            GVL_EVENT.G_Event_Log[GVL_EVENT.G_Event_Head].Event_ID := GVL_EVENT.G_Event_ID_Counter;
GVL_EVENT.G_Event_Log[GVL_EVENT.G_Event_Head].Event_Type := VI_Event_Type;
GVL_EVENT.G_Event_Log[GVL_EVENT.G_Event_Head].Timestamp := VI_Timestamp;
GVL_EVENT.G_Event_Log[GVL_EVENT.G_Event_Head].Param1 := VI_Param1;
GVL_EVENT.G_Event_Log[GVL_EVENT.G_Event_Head].Param2 := VI_Param2;

GVL_EVENT.G_Event_ID_Counter := GVL_EVENT.G_Event_ID_Counter + 1;
GVL_EVENT.G_Event_Head := (GVL_EVENT.G_Event_Head + 1) MOD 64;
          
END_FUNCTION_BLOCK

FUNCTION_BLOCK FB_Fault_Logger
  VAR_INPUT
    VI_Severity : E_System_Severity;
    VI_RootCause : E_System_Root_Cause;
    VI_Time_MS : UDINT;
  END_VAR
  VAR_OUTPUT
    VO_Last_Event_Text : STRING(200);
    VO_Event_Count : UINT;
    VO_Last_Index : UINT;
    VO_Event_Time_MS : ARRAY[1..16] OF UDINT;
    VO_Event_Severity : ARRAY[1..16] OF E_System_Severity;
    VO_Event_RootCause : ARRAY[1..16] OF E_System_Root_Cause;
    VO_Event_Text : ARRAY[1..16] OF STRING(200);
  END_VAR
  VAR
    L_Last_Severity : E_System_Severity;
    L_Last_RootCause : E_System_Root_Cause;
    L_Write_Index : UINT := 0;
    L_Event_Text : STRING(200);
  END_VAR

            L_Event_Text := '';

IF (VI_Severity <> L_Last_Severity) OR (VI_RootCause <> L_Last_RootCause) THEN
    CASE VI_RootCause OF
        E_System_Root_Cause.ROOT_FIRE:
            L_Event_Text := 'EVENT: FIRE DETECTED';
        E_System_Root_Cause.ROOT_GAS_LEAK:
            L_Event_Text := 'EVENT: GAS LEAK';
        E_System_Root_Cause.ROOT_CO_CRITICAL:
            L_Event_Text := 'EVENT: CO CRITICAL';
        E_System_Root_Cause.ROOT_CO_WARNING:
            L_Event_Text := 'EVENT: CO WARNING';
        E_System_Root_Cause.ROOT_WATER_LEAK:
            L_Event_Text := 'EVENT: WATER LEAK';
        E_System_Root_Cause.ROOT_SENSOR_FAULT:
            L_Event_Text := 'EVENT: SENSOR FAULT';
        E_System_Root_Cause.ROOT_IO_OFFLINE:
            L_Event_Text := 'EVENT: IO OFFLINE';
        E_System_Root_Cause.ROOT_COMM_FAULT:
            L_Event_Text := 'EVENT: COMM FAULT';
        E_System_Root_Cause.ROOT_WATCHDOG_FAULT:
            L_Event_Text := 'EVENT: WATCHDOG FAULT';
        E_System_Root_Cause.ROOT_SUBSYSTEM_FAULT:
            L_Event_Text := 'EVENT: SUBSYSTEM FAULT';
        ELSE
            L_Event_Text := 'EVENT: SYSTEM STATE CHANGE';
    END_CASE;

    L_Write_Index := L_Write_Index + 1;
    IF L_Write_Index > 16 THEN
        L_Write_Index := 1;
    END_IF;

    VO_Event_Time_MS[L_Write_Index] := VI_Time_MS;
    VO_Event_Severity[L_Write_Index] := VI_Severity;
    VO_Event_RootCause[L_Write_Index] := VI_RootCause;
    VO_Event_Text[L_Write_Index] := L_Event_Text;

    VO_Last_Index := L_Write_Index;
    VO_Last_Event_Text := L_Event_Text;

    IF VO_Event_Count < 16 THEN
        VO_Event_Count := VO_Event_Count + 1;
    END_IF;
END_IF;

L_Last_Severity := VI_Severity;
L_Last_RootCause := VI_RootCause;
// >>> BULK_SYNC_ANCHOR: FB_Fault_Logger <<<
          
END_FUNCTION_BLOCK

FUNCTION_BLOCK FB_CoreKernel_Live_Observer

            
          
END_FUNCTION_BLOCK

FUNCTION_BLOCK FB_FloorHeating_Overheat_Protection
  VAR_INPUT
    VI_Threshold : REAL := 45.0;
  END_VAR
  VAR_OUTPUT
    VO_Overheat_Detected : BOOL;
    VO_Locked_Circuits : ARRAY[1..GVL_CONSTANTS.C_MAX_HEATING_CIRCUITS] OF BOOL;
  END_VAR
  VAR_IN_OUT
    VI_Temps : ARRAY[1..GVL_CONSTANTS.C_MAX_HEATING_CIRCUITS] OF REAL;
  END_VAR
  VAR
    L_i : INT;
  END_VAR

            VO_Overheat_Detected := FALSE;
FOR L_i := 1 TO GVL_CONSTANTS.C_MAX_HEATING_CIRCUITS DO
    IF VI_Temps[L_i] > VI_Threshold THEN
        VO_Overheat_Detected := TRUE;
        VO_Locked_Circuits[L_i] := TRUE;
    END_IF;
END_FOR;
          
END_FUNCTION_BLOCK

FUNCTION_BLOCK FB_HMI_Interface
  VAR_INPUT
    VI_Severity : E_System_Severity;
    VI_RootCause : E_System_Root_Cause;
    VI_Status_Msg : STRING(200);
  END_VAR
  VAR_OUTPUT
    VO_HMI_Status_Text : STRING(200);
    VO_HMI_State_Code : INT;
  END_VAR

            VO_HMI_Status_Text := VI_Status_Msg;

CASE VI_Severity OF
    E_System_Severity.SEV_NORMAL:
        VO_HMI_State_Code := 0;
    E_System_Severity.SEV_WARNING:
        VO_HMI_State_Code := 1;
    E_System_Severity.SEV_DEGRADED:
        VO_HMI_State_Code := 2;
    E_System_Severity.SEV_CRITICAL:
        VO_HMI_State_Code := 3;
END_CASE;
// >>> BULK_SYNC_ANCHOR: FB_HMI_Interface <<<
          
END_FUNCTION_BLOCK

FUNCTION_BLOCK FB_System_Health
  VAR_INPUT
    VI_Smoke_Detected : BOOL;
    VI_Gas_Detected : BOOL;
    VI_CO_Warning_Level : BOOL;
    VI_CO_Alarm_Level : BOOL;
    VI_Leak_Detected : BOOL;
    VI_Sensor_Fault : BOOL := FALSE;
    VI_IO_Offline : BOOL := FALSE;
    VI_Comm_Fault : BOOL := FALSE;
    VI_Watchdog_Fault : BOOL := FALSE;
    VI_Subsystem_Fault : BOOL := FALSE;
  END_VAR
  VAR_OUTPUT
    VO_System_Severity : E_System_Severity;
    VO_Root_Cause : E_System_Root_Cause;
    VO_Sensor_Fault : BOOL;
    VO_IO_Fault : BOOL;
    VO_Comm_Fault : BOOL;
    VO_Subsystem_Degraded : BOOL;
    VO_First_Fault_Active : BOOL;
    VO_First_Fault_Type : INT;
    VO_First_Fault_Source : INT;
    VO_IO_Fault_Count : UDINT;
    VO_Comm_Fault_Count : UDINT;
    VO_Sensor_Fault_Count : UDINT;
    VO_Subsystem_Fault_Count : UDINT;
    VO_Watchdog_Fault_Count : UDINT;
  END_VAR
  VAR
    L_IO_Fault_Assert_Count : UINT;
    L_IO_Fault_Clear_Count : UINT;
    L_IO_Fault_Stable : BOOL;
    L_Comm_Fault_Assert_Count : UINT;
    L_Comm_Fault_Clear_Count : UINT;
    L_Comm_Fault_Stable : BOOL;
    L_Sensor_Fault_Assert_Count : UINT;
    L_Sensor_Fault_Clear_Count : UINT;
    L_Sensor_Fault_Stable : BOOL;
    L_Subsystem_Assert_Count : UINT;
    L_Subsystem_Clear_Count : UINT;
    L_Subsystem_Fault_Stable : BOOL;
    L_IO_Fault_Prev : BOOL;
    L_Comm_Fault_Prev : BOOL;
    L_Sensor_Fault_Prev : BOOL;
    L_Subsystem_Fault_Prev : BOOL;
    L_Watchdog_Fault_Prev : BOOL;
  END_VAR
  VAR CONSTANT
    C_HEALTH_DEBOUNCE_CYCLES : UINT := 3;
  END_VAR

            // Debounce non-critical diagnostics: require 3 stable cycles to assert/clear
IF VI_IO_Offline THEN
    L_IO_Fault_Clear_Count := 0;
    IF L_IO_Fault_Assert_Count < C_HEALTH_DEBOUNCE_CYCLES THEN
        L_IO_Fault_Assert_Count := L_IO_Fault_Assert_Count + 1;
    END_IF;
    IF L_IO_Fault_Assert_Count >= C_HEALTH_DEBOUNCE_CYCLES THEN
        L_IO_Fault_Stable := TRUE;
    END_IF;
ELSE
    L_IO_Fault_Assert_Count := 0;
    IF L_IO_Fault_Clear_Count < C_HEALTH_DEBOUNCE_CYCLES THEN
        L_IO_Fault_Clear_Count := L_IO_Fault_Clear_Count + 1;
    END_IF;
    IF L_IO_Fault_Clear_Count >= C_HEALTH_DEBOUNCE_CYCLES THEN
        L_IO_Fault_Stable := FALSE;
    END_IF;
END_IF;

IF VI_Comm_Fault THEN
    L_Comm_Fault_Clear_Count := 0;
    IF L_Comm_Fault_Assert_Count < C_HEALTH_DEBOUNCE_CYCLES THEN
        L_Comm_Fault_Assert_Count := L_Comm_Fault_Assert_Count + 1;
    END_IF;
    IF L_Comm_Fault_Assert_Count >= C_HEALTH_DEBOUNCE_CYCLES THEN
        L_Comm_Fault_Stable := TRUE;
    END_IF;
ELSE
    L_Comm_Fault_Assert_Count := 0;
    IF L_Comm_Fault_Clear_Count < C_HEALTH_DEBOUNCE_CYCLES THEN
        L_Comm_Fault_Clear_Count := L_Comm_Fault_Clear_Count + 1;
    END_IF;
    IF L_Comm_Fault_Clear_Count >= C_HEALTH_DEBOUNCE_CYCLES THEN
        L_Comm_Fault_Stable := FALSE;
    END_IF;
END_IF;

IF VI_Sensor_Fault THEN
    L_Sensor_Fault_Clear_Count := 0;
    IF L_Sensor_Fault_Assert_Count < C_HEALTH_DEBOUNCE_CYCLES THEN
        L_Sensor_Fault_Assert_Count := L_Sensor_Fault_Assert_Count + 1;
    END_IF;
    IF L_Sensor_Fault_Assert_Count >= C_HEALTH_DEBOUNCE_CYCLES THEN
        L_Sensor_Fault_Stable := TRUE;
    END_IF;
ELSE
    L_Sensor_Fault_Assert_Count := 0;
    IF L_Sensor_Fault_Clear_Count < C_HEALTH_DEBOUNCE_CYCLES THEN
        L_Sensor_Fault_Clear_Count := L_Sensor_Fault_Clear_Count + 1;
    END_IF;
    IF L_Sensor_Fault_Clear_Count >= C_HEALTH_DEBOUNCE_CYCLES THEN
        L_Sensor_Fault_Stable := FALSE;
    END_IF;
END_IF;

IF VI_Subsystem_Fault THEN
    L_Subsystem_Clear_Count := 0;
    IF L_Subsystem_Assert_Count < C_HEALTH_DEBOUNCE_CYCLES THEN
        L_Subsystem_Assert_Count := L_Subsystem_Assert_Count + 1;
    END_IF;
    IF L_Subsystem_Assert_Count >= C_HEALTH_DEBOUNCE_CYCLES THEN
        L_Subsystem_Fault_Stable := TRUE;
    END_IF;
ELSE
    L_Subsystem_Assert_Count := 0;
    IF L_Subsystem_Clear_Count < C_HEALTH_DEBOUNCE_CYCLES THEN
        L_Subsystem_Clear_Count := L_Subsystem_Clear_Count + 1;
    END_IF;
    IF L_Subsystem_Clear_Count >= C_HEALTH_DEBOUNCE_CYCLES THEN
        L_Subsystem_Fault_Stable := FALSE;
    END_IF;
END_IF;

// Count confirmed fault events on rising edge of stable/critical conditions
IF L_IO_Fault_Stable AND NOT L_IO_Fault_Prev THEN
    VO_IO_Fault_Count := VO_IO_Fault_Count + 1;
END_IF;
L_IO_Fault_Prev := L_IO_Fault_Stable;

IF L_Comm_Fault_Stable AND NOT L_Comm_Fault_Prev THEN
    VO_Comm_Fault_Count := VO_Comm_Fault_Count + 1;
END_IF;
L_Comm_Fault_Prev := L_Comm_Fault_Stable;

IF L_Sensor_Fault_Stable AND NOT L_Sensor_Fault_Prev THEN
    VO_Sensor_Fault_Count := VO_Sensor_Fault_Count + 1;
END_IF;
L_Sensor_Fault_Prev := L_Sensor_Fault_Stable;

IF L_Subsystem_Fault_Stable AND NOT L_Subsystem_Fault_Prev THEN
    VO_Subsystem_Fault_Count := VO_Subsystem_Fault_Count + 1;
END_IF;
L_Subsystem_Fault_Prev := L_Subsystem_Fault_Stable;

IF VI_Watchdog_Fault AND NOT L_Watchdog_Fault_Prev THEN
    VO_Watchdog_Fault_Count := VO_Watchdog_Fault_Count + 1;
END_IF;
L_Watchdog_Fault_Prev := VI_Watchdog_Fault;

VO_Sensor_Fault := L_Sensor_Fault_Stable;
VO_IO_Fault := L_IO_Fault_Stable;
VO_Comm_Fault := L_Comm_Fault_Stable;
VO_Subsystem_Degraded := L_Subsystem_Fault_Stable;

VO_System_Severity := E_System_Severity.SEV_NORMAL;
VO_Root_Cause := E_System_Root_Cause.ROOT_NONE;
VO_First_Fault_Active := FALSE;
VO_First_Fault_Type := 0;
VO_First_Fault_Source := 0;

// Priority: FIRE > GAS > CO > WATER > diagnostics
IF VI_Smoke_Detected THEN
    VO_System_Severity := E_System_Severity.SEV_CRITICAL;
    VO_Root_Cause := E_System_Root_Cause.ROOT_FIRE;
    VO_First_Fault_Active := TRUE;
    VO_First_Fault_Type := 5;

ELSIF VI_Gas_Detected THEN
    VO_System_Severity := E_System_Severity.SEV_CRITICAL;
    VO_Root_Cause := E_System_Root_Cause.ROOT_GAS_LEAK;
    VO_First_Fault_Active := TRUE;
    VO_First_Fault_Type := 6;

ELSIF VI_CO_Alarm_Level THEN
    VO_System_Severity := E_System_Severity.SEV_CRITICAL;
    VO_Root_Cause := E_System_Root_Cause.ROOT_CO_CRITICAL;
    VO_First_Fault_Active := TRUE;
    VO_First_Fault_Type := 7;

ELSIF VI_CO_Warning_Level THEN
    VO_System_Severity := E_System_Severity.SEV_WARNING;
    VO_Root_Cause := E_System_Root_Cause.ROOT_CO_WARNING;
    VO_First_Fault_Active := TRUE;
    VO_First_Fault_Type := 7;

ELSIF VI_Leak_Detected THEN
    VO_System_Severity := E_System_Severity.SEV_WARNING;
    VO_Root_Cause := E_System_Root_Cause.ROOT_WATER_LEAK;
    VO_First_Fault_Active := TRUE;
    VO_First_Fault_Type := 8;

ELSIF VI_Watchdog_Fault THEN
    VO_System_Severity := E_System_Severity.SEV_CRITICAL;
    VO_Root_Cause := E_System_Root_Cause.ROOT_WATCHDOG_FAULT;
    VO_First_Fault_Active := TRUE;
    VO_First_Fault_Type := 9;

ELSIF L_IO_Fault_Stable THEN
    VO_System_Severity := E_System_Severity.SEV_DEGRADED;
    VO_Root_Cause := E_System_Root_Cause.ROOT_IO_OFFLINE;
    VO_First_Fault_Active := TRUE;
    VO_First_Fault_Type := 1;

ELSIF L_Comm_Fault_Stable THEN
    VO_System_Severity := E_System_Severity.SEV_DEGRADED;
    VO_Root_Cause := E_System_Root_Cause.ROOT_COMM_FAULT;
    VO_First_Fault_Active := TRUE;
    VO_First_Fault_Type := 3;

ELSIF L_Sensor_Fault_Stable THEN
    VO_System_Severity := E_System_Severity.SEV_DEGRADED;
    VO_Root_Cause := E_System_Root_Cause.ROOT_SENSOR_FAULT;
    VO_First_Fault_Active := TRUE;
    VO_First_Fault_Type := 2;

ELSIF L_Subsystem_Fault_Stable THEN
    VO_System_Severity := E_System_Severity.SEV_DEGRADED;
    VO_Root_Cause := E_System_Root_Cause.ROOT_SUBSYSTEM_FAULT;
    VO_First_Fault_Active := TRUE;
    VO_First_Fault_Type := 4;
END_IF;
// >>> BULK_SYNC_ANCHOR: FB_System_Health <<<
          
END_FUNCTION_BLOCK

FUNCTION_BLOCK FB_Lifetime_Predictor
  VAR_INPUT
    VI_Runtime_Hours : UDINT;
    VI_Start_Count : UDINT;
    VI_Nominal_Life : UDINT := 10000;
  END_VAR
  VAR_OUTPUT
    VO_Remaining_Percent : BYTE;
    VO_Maintenance_Req : BOOL;
  END_VAR

            // Упрощенная модель износа
IF VI_Nominal_Life > 0 THEN
    VO_Remaining_Percent := TO_BYTE(100 - (VI_Runtime_Hours * 100 / VI_Nominal_Life));
ELSE
    VO_Remaining_Percent := 0;
END_IF;

VO_Maintenance_Req := (VO_Remaining_Percent < 10);
          
END_FUNCTION_BLOCK

FUNCTION_BLOCK FB_Persist_Pipeline
  VAR_INPUT
    VI_PersistStruct : ST_Persist;
    VI_System_Time_MS : UDINT;
    VI_IsActivePLC : BOOL;
  END_VAR
  VAR_OUTPUT
    VO_NVRAM_Cmd : BYTE;
    VO_NVRAM_Offset : UDINT;
    VO_NVRAM_Done : BOOL;
    VO_NVRAM_Err : BOOL;
    VO_NVRAM_ErrID : UDINT;
  END_VAR
  VAR_IN_OUT
    VIO_Apply_Settings : BOOL;
    VIO_Persist_Buffer : ARRAY[0..4] OF BYTE;
    VIO_Last_Written_Persist_Buffer : ARRAY[0..4] OF BYTE;
    VIO_Last_Persist_Write_MS : UDINT;
  END_VAR
  VAR
    fbNVRAMManager : FB_NVRAM_Manager;
    L_Persist_Buffer_Changed : BOOL;
  END_VAR

            // === SERIALIZE PERSIST STRUCT → BUFFER ===

// System Mode
VIO_Persist_Buffer[0] := TO_BYTE(TO_INT(VI_PersistStruct.System_Mode));

// Gas
IF VI_PersistStruct.Safety_Gas_Latched THEN
    VIO_Persist_Buffer[1] := BYTE#1;
ELSE
    VIO_Persist_Buffer[1] := BYTE#0;
END_IF;

// Smoke
IF VI_PersistStruct.Safety_Smoke_Latched THEN
    VIO_Persist_Buffer[2] := BYTE#1;
ELSE
    VIO_Persist_Buffer[2] := BYTE#0;
END_IF;

// Leak
IF VI_PersistStruct.Safety_Leak_Latched THEN
    VIO_Persist_Buffer[3] := BYTE#1;
ELSE
    VIO_Persist_Buffer[3] := BYTE#0;
END_IF;

// DHW Pump
IF VI_PersistStruct.DHW_Heating_Pump THEN
    VIO_Persist_Buffer[4] := BYTE#1;
ELSE
    VIO_Persist_Buffer[4] := BYTE#0;
END_IF;

// === END SERIALIZE ===

L_Persist_Buffer_Changed :=
    (VIO_Persist_Buffer[0] <> VIO_Last_Written_Persist_Buffer[0]) OR
    (VIO_Persist_Buffer[1] <> VIO_Last_Written_Persist_Buffer[1]) OR
    (VIO_Persist_Buffer[2] <> VIO_Last_Written_Persist_Buffer[2]) OR
    (VIO_Persist_Buffer[3] <> VIO_Last_Written_Persist_Buffer[3]) OR
    (VIO_Persist_Buffer[4] <> VIO_Last_Written_Persist_Buffer[4]);

VO_NVRAM_Cmd := 0;
VO_NVRAM_Offset := 0;

IF VIO_Apply_Settings THEN
    // explicit config apply requests a controlled write
    // keep flag set until successful write confirmation
    VO_NVRAM_Cmd := 1;

ELSIF L_Persist_Buffer_Changed THEN
    // controlled write: no more often than once per 60 seconds
    IF (VIO_Last_Persist_Write_MS = 0) OR
       ((VI_System_Time_MS - VIO_Last_Persist_Write_MS) >= 60000) THEN
        VO_NVRAM_Cmd := 1;
    END_IF;
END_IF;

fbNVRAMManager(
    VI_Command := VO_NVRAM_Cmd,
    VI_Offset := VO_NVRAM_Offset,
    VI_DataRef := VIO_Persist_Buffer[0],
    VI_DataSize := 5,
    VI_System_Time_MS := VI_System_Time_MS,
    VI_Operator_ID := 'SYSTEM',
    VI_IsActivePLC := VI_IsActivePLC,
    VI_TwoPersonConfirmation := FALSE,
    VO_Done => VO_NVRAM_Done,
    VO_Error => VO_NVRAM_Err,
    VO_ErrorID => VO_NVRAM_ErrID
);

IF (VO_NVRAM_Cmd = 1) AND VO_NVRAM_Done AND NOT VO_NVRAM_Err THEN
    VIO_Last_Written_Persist_Buffer[0] := VIO_Persist_Buffer[0];
    VIO_Last_Written_Persist_Buffer[1] := VIO_Persist_Buffer[1];
    VIO_Last_Written_Persist_Buffer[2] := VIO_Persist_Buffer[2];
    VIO_Last_Written_Persist_Buffer[3] := VIO_Persist_Buffer[3];
    VIO_Last_Written_Persist_Buffer[4] := VIO_Persist_Buffer[4];
    VIO_Last_Persist_Write_MS := VI_System_Time_MS;
    VIO_Apply_Settings := FALSE;
END_IF;
          
END_FUNCTION_BLOCK

FUNCTION_BLOCK FB_Trend_Adapter
  VAR_INPUT
    VI_Data : ST_Trend_Data;
  END_VAR
  VAR_OUTPUT
    VO_Average : REAL;
    VO_Min : REAL;
    VO_Max : REAL;
    VO_Trend_Up : BOOL;
    VO_Trend_Down : BOOL;
  END_VAR
  VAR
    fbAnalyzer : FB_Trend_Analyzer;
    L_Data_Copy : ARRAY[1..GVL_CONSTANTS.C_MAX_TREND_DATA_POINTS] OF REAL;
    L_Count : INT;
    L_i : INT;
  END_VAR

            // Normalize count to analyzer bounds
L_Count := UDINT_TO_INT(VI_Data.record_count);
IF L_Count < 0 THEN
    L_Count := 0;
END_IF;
IF L_Count > GVL_CONSTANTS.C_MAX_TREND_DATA_POINTS THEN
    L_Count := GVL_CONSTANTS.C_MAX_TREND_DATA_POINTS;
END_IF;

// Copy source values into analyzer-compatible buffer
FOR L_i := 1 TO GVL_CONSTANTS.C_MAX_TREND_DATA_POINTS DO
    L_Data_Copy[L_i] := 0.0;
END_FOR;

IF L_Count > 0 THEN
    FOR L_i := 1 TO L_Count DO
        L_Data_Copy[L_i] := VI_Data.values[L_i];
    END_FOR;
END_IF;

fbAnalyzer(
    VI_Count := L_Count,
    VI_Data := L_Data_Copy,
    VO_Average => VO_Average,
    VO_Max => VO_Max,
    VO_Min => VO_Min,
    VO_Trend_Up => VO_Trend_Up,
    VO_Trend_Down => VO_Trend_Down
);
          
END_FUNCTION_BLOCK

FUNCTION_BLOCK FB_System_Redundancy_Orchestrator
  VAR_IN_OUT
    VIO_Local_State : ST_System_State_Snapshot;
    VIO_Remote_State : ST_System_State_Snapshot;
  END_VAR
  VAR
    fbRedundancy : FB_Redundancy_Manager;
  END_VAR

            // ==============================================================================
// System redundancy orchestrator helper
//
// Internal helper for PRG_System.
// Owns PLC role calculation, heartbeat output projection, and synced-state apply.
// ==============================================================================



// Build local state snapshot for replication.
VIO_Local_State.System_Time_MS := GVL_STATUS.G_System_Time_MS;
VIO_Local_State.Current_Scenario := GVL_STATUS.G_Current_Scenario;
VIO_Local_State.Security_Armed := GVL_ALARM.G_Security_Armed;
VIO_Local_State.Active_Alarms := GVL_ALARM.G_Active_Alarm_Count;
VIO_Local_State.Zone_Valves := GVL_STATE.G_Zone_Valves;
VIO_Local_State.Manifold_Pumps := GVL_STATE.G_Manifold_Pumps;
VIO_Local_State.Lighting_States := GVL_STATE.G_Lighting_Levels;
VIO_Local_State.Blinds_Positions := GVL_STATE.G_Blinds_Positions;
VIO_Local_State.Socket_States := GVL_STATE.G_Socket_States;
VIO_Local_State.Gas_Valve_Closed := GVL_COMMAND.G_Gas_Valve_Close;
VIO_Local_State.Water_Valves_Closed := GVL_COMMAND.G_Close_Valve_36;
VIO_Local_State.Version := VIO_Local_State.Version + 1;

fbRedundancy(
    VI_System_Time_MS := GVL_STATUS.G_System_Time_MS,
    VI_Local_PLC_ID := GVL_STATUS.G_PLC_ID,
    VI_Remote_Pulse := GVL_IO.DI_Partner_Pulse,
    VI_Remote_Is_Active := GVL_IO.DI_Partner_Active,
    VI_Gateway_Ping_OK := GVL_GATEWAY.G_Gateway_Ping_OK,
    VI_Local_State := VIO_Local_State,
    VI_Remote_State := VIO_Remote_State
);

GVL_STATUS.G_Is_Active_PLC := (fbRedundancy.VO_Local_Role = E_PLC_ROLE.ROLE_ACTIVE);
GVL_IO.DO_Heartbeat_Pulse := fbRedundancy.VO_Local_Pulse;
GVL_IO.DO_Active_Status := GVL_STATUS.G_Is_Active_PLC;

IF fbRedundancy.VO_State_Updated THEN
    GVL_STATUS.G_Current_Scenario := fbRedundancy.VO_Synced_State.Current_Scenario;
    GVL_ALARM.G_Security_Armed := fbRedundancy.VO_Synced_State.Security_Armed;
    GVL_STATE.G_Zone_Valves := fbRedundancy.VO_Synced_State.Zone_Valves;
    GVL_STATE.G_Manifold_Pumps := fbRedundancy.VO_Synced_State.Manifold_Pumps;
    GVL_STATE.G_Lighting_Levels := fbRedundancy.VO_Synced_State.Lighting_States;
    GVL_STATE.G_Blinds_Positions := fbRedundancy.VO_Synced_State.Blinds_Positions;
    GVL_STATE.G_Socket_States := fbRedundancy.VO_Synced_State.Socket_States;
    GVL_COMMAND.G_Gas_Valve_Close := fbRedundancy.VO_Synced_State.Gas_Valve_Closed;
    GVL_COMMAND.G_Close_Valve_36 := fbRedundancy.VO_Synced_State.Water_Valves_Closed;
    VIO_Local_State.Version := fbRedundancy.VO_Synced_State.Version;
END_IF;

// >>> BULK_SYNC_ANCHOR: FB_System_Redundancy_Orchestrator <<<
          
END_FUNCTION_BLOCK

FUNCTION_BLOCK FB_Diagnostics_Event_Manager
  VAR_INPUT
    VI_Code : UDINT;
    VI_Severity : INT;
    VI_Active : BOOL;
    VI_Timestamp : UDINT;
    VI_Source : INT;
  END_VAR
  VAR_IN_OUT
    VIO_Events : ARRAY[1..50] OF ST_Diagnostic_Event;
    VIO_Count : INT;
  END_VAR
  VAR
    L_i : INT;
    L_Found_Index : INT;
    L_Was_Active : BOOL;
  END_VAR

            L_Found_Index := 0;
L_Was_Active := FALSE;

FOR L_i := 1 TO VIO_Count DO
    IF (VIO_Events[L_i].Code = VI_Code) AND (VIO_Events[L_i].Source = VI_Source) THEN
        L_Found_Index := L_i;
        L_Was_Active := VIO_Events[L_i].Active;
    END_IF;
END_FOR;

IF VI_Active THEN
    IF L_Found_Index = 0 THEN
        IF VIO_Count < 50 THEN
            VIO_Count := VIO_Count + 1;
            VIO_Events[VIO_Count].Code := VI_Code;
            VIO_Events[VIO_Count].Severity := VI_Severity;
            VIO_Events[VIO_Count].Active := TRUE;
            VIO_Events[VIO_Count].Timestamp := VI_Timestamp;
            VIO_Events[VIO_Count].Source := VI_Source;
        END_IF;
    ELSE
        VIO_Events[L_Found_Index].Severity := VI_Severity;
        IF NOT L_Was_Active THEN
            VIO_Events[L_Found_Index].Timestamp := VI_Timestamp;
        END_IF;
        VIO_Events[L_Found_Index].Active := TRUE;
    END_IF;
ELSE
    IF L_Found_Index > 0 THEN
        VIO_Events[L_Found_Index].Active := FALSE;
    END_IF;
END_IF;
          
END_FUNCTION_BLOCK

FUNCTION_BLOCK FB_Access_Control
  VAR_INPUT
    VI_System_Time_MS : UDINT;
    VI_IsActivePLC : BOOL;
    VI_Armed : BOOL;
    VI_System_Mode : E_System_Operating_Mode;
    VI_Gate_Open_Req : BOOL;
    VI_Wicket_Open_Req : BOOL;
    VI_Lock_1_Open_Req : BOOL;
    VI_Lock_1_Close_Req : BOOL;
    VI_Lock_2_Open_Req : BOOL;
    VI_Lock_2_Close_Req : BOOL;
    VI_PIN_Code : STRING(4);
    VI_RFID_Tag : STRING(20);
    VI_Config : ST_Security_Global_Config;
  END_VAR
  VAR_OUTPUT
    VO_Gate_Open : BOOL;
    VO_Wicket_Open : BOOL;
    VO_Lock_1_Open : BOOL;
    VO_Lock_1_Close : BOOL;
    VO_Lock_2_Open : BOOL;
    VO_Lock_2_Close : BOOL;
  END_VAR
  VAR_IN_OUT
    VI_Access_Codes : ARRAY[1..GVL_CONSTANTS.C_MAX_ACCESS_CODES] OF DWORD;
    VI_RFID_Tags : ARRAY[1..GVL_CONSTANTS.C_MAX_ACCESS_CODES] OF STRING(20);
  END_VAR
  VAR
    L_Gate_Timer : TP;
    L_Wicket_Timer : TP;
    L_Lock_1_Open_T : TP;
    L_Lock_1_Close_T : TP;
    L_Lock_2_Open_T : TP;
    L_Lock_2_Close_T : TP;
    L_Prev_Armed : BOOL;
    L_Auto_Lock_Req : BOOL;
    R_Trig_Gate : R_TRIG;
    R_Trig_Wicket : R_TRIG;
    R_Trig_Lock_1_O : R_TRIG;
    R_Trig_Lock_1_C : R_TRIG;
    R_Trig_Lock_2_O : R_TRIG;
    R_Trig_Lock_2_C : R_TRIG;
    fbAccessCode : FB_AccessCode_Manager;
    L_Valid_PIN : BOOL;
  END_VAR

            // Если ПЛК находится в режиме Standby (резерв), он не должен управлять выходами
IF NOT VI_IsActivePLC THEN
    RETURN;
END_IF;

IF VI_System_Mode = E_System_Operating_Mode.MODE_SAFE_STOP THEN
    VO_Gate_Open := FALSE;
    VO_Wicket_Open := FALSE;
    VO_Lock_1_Open := FALSE;
    VO_Lock_2_Open := FALSE;
    RETURN;
END_IF;

// 1. Логика автоматического закрытия замков при постановке на охрану (ТЗ 3.0)
// При переходе системы в режим "Охрана" принудительно блокируем все замки
IF VI_Armed AND NOT L_Prev_Armed THEN
    L_Auto_Lock_Req := TRUE;
END_IF;
L_Prev_Armed := VI_Armed;

// Детекторы фронта для команд
R_Trig_Gate(CLK := VI_Gate_Open_Req);
R_Trig_Wicket(CLK := VI_Wicket_Open_Req);
R_Trig_Lock_1_O(CLK := VI_Lock_1_Open_Req);
R_Trig_Lock_1_C(CLK := VI_Lock_1_Close_Req OR L_Auto_Lock_Req);
R_Trig_Lock_2_O(CLK := VI_Lock_2_Open_Req);
R_Trig_Lock_2_C(CLK := VI_Lock_2_Close_Req OR L_Auto_Lock_Req);

// Проверка PIN-кода или RFID-метки через менеджер кодов
fbAccessCode(
    VI_System_Time_MS := VI_System_Time_MS,
    VI_IsActivePLC := VI_IsActivePLC,
    VI_Code_To_Check := VI_PIN_Code,
    VI_RFID_To_Check := VI_RFID_Tag,
    VI_Access_Codes := VI_Access_Codes,
    VI_RFID_Tags := VI_RFID_Tags,
    VO_Code_Valid => L_Valid_PIN
);

// 2. Формирование импульсов управления исполнительными механизмами (Pulse Control)
// Открытие ворот и калитки требует валидного ПИН-кода или RFID-метки, если система под охраной
L_Gate_Timer(IN := R_Trig_Gate.Q AND (NOT VI_Armed OR L_Valid_PIN), PT := TO_TIME(VI_Config.gate_open_pulse_ms));
VO_Gate_Open := L_Gate_Timer.Q;

L_Wicket_Timer(IN := R_Trig_Wicket.Q AND (NOT VI_Armed OR L_Valid_PIN), PT := TO_TIME(VI_Config.wicket_open_pulse_ms));
VO_Wicket_Open := L_Wicket_Timer.Q;

L_Lock_1_Open_T(IN := R_Trig_Lock_1_O.Q AND (NOT VI_Armed OR L_Valid_PIN), PT := TO_TIME(VI_Config.lock_open_pulse_ms));
VO_Lock_1_Open := L_Lock_1_Open_T.Q;

L_Lock_1_Close_T(IN := R_Trig_Lock_1_C.Q, PT := TO_TIME(VI_Config.lock_close_pulse_ms));
VO_Lock_1_Close := L_Lock_1_Close_T.Q;

L_Lock_2_Open_T(IN := R_Trig_Lock_2_O.Q AND (NOT VI_Armed OR L_Valid_PIN), PT := TO_TIME(VI_Config.lock_open_pulse_ms));
VO_Lock_2_Open := L_Lock_2_Open_T.Q;

L_Lock_2_Close_T(IN := R_Trig_Lock_2_C.Q, PT := TO_TIME(VI_Config.lock_close_pulse_ms));
VO_Lock_2_Close := L_Lock_2_Close_T.Q;

// Сброс флага автоматического закрытия
IF L_Auto_Lock_Req THEN
    L_Auto_Lock_Req := FALSE;
END_IF;
// >>> BULK_SYNC_ANCHOR: FB_Access_Control <<<
          
END_FUNCTION_BLOCK

FUNCTION_BLOCK FB_Trend_Logger
  VAR_INPUT
    VI_System_Time_MS : UDINT;
    VI_Config : ST_Trend_Config;
    VI_Current_Value : REAL;
  END_VAR
  VAR_OUTPUT
    VO_Data : ST_Trend_Data;
  END_VAR
  VAR
    L_Last_Log_Time : UDINT;
    L_Last_Value : REAL;
    L_Deviation : REAL;
  END_VAR

            IF NOT VI_Config.enabled THEN RETURN; END_IF;

// Логирование по изменению (Deadband) или по времени (раз в час)
L_Deviation := ABS(VI_Current_Value - L_Last_Value);
IF (L_Deviation >= (L_Last_Value * VI_Config.deviation_threshold_percent / 100.0)) OR 
   ((SEL(VI_System_Time_MS >= L_Last_Log_Time, VI_System_Time_MS - L_Last_Log_Time, (4294967295 - L_Last_Log_Time) + VI_System_Time_MS + 1)) >= GVL_CONSTANTS.C_MS_IN_HOUR) THEN
    
    // Запись в массив
    VO_Data.write_index := (VO_Data.record_count MOD 100) + 1;
    VO_Data.values[VO_Data.write_index] := VI_Current_Value;
    VO_Data.timestamps[VO_Data.write_index] := VI_System_Time_MS;

    VO_Data.record_count := VO_Data.record_count + 1;
    VO_Data.sum_values := VO_Data.sum_values + VI_Current_Value;
    
    L_Last_Value := VI_Current_Value;
    L_Last_Log_Time := VI_System_Time_MS;
END_IF;
          
END_FUNCTION_BLOCK

FUNCTION_BLOCK FB_State_Trace_Log
  VAR_INPUT
    VI_System_Time : UDINT;
    VI_Gas_Alarm : BOOL;
    VI_Leak_Alarm : BOOL;
    VI_Pumps : ARRAY[1..4] OF BOOL;
  END_VAR
  VAR_OUTPUT
    VO_Last_Change_Time : UDINT;
  END_VAR
  VAR
    L_Last_Gas : BOOL;
    L_Last_Leak : BOOL;
  END_VAR

            IF (VI_Gas_Alarm <> L_Last_Gas) OR (VI_Leak_Alarm <> L_Last_Leak) THEN
    VO_Last_Change_Time := VI_System_Time;
END_IF;

L_Last_Gas := VI_Gas_Alarm;
L_Last_Leak := VI_Leak_Alarm;
          
END_FUNCTION_BLOCK

FUNCTION_BLOCK FB_System_Timer
  VAR_INPUT
    IN : BOOL;
    PT : TIME;
    VI_System_Time_MS : UDINT;
  END_VAR
  VAR_OUTPUT
    Q : BOOL;
    ET : TIME;
  END_VAR
  VAR
    L_Start_Time : UDINT;
    L_Running : BOOL;
  END_VAR

            // ==============================================================================
// Блок таймера, привязанный к системному времени (System Timer)
// Назначение:
// - Замена стандартного TON для обеспечения точной выдержки времени,
//   независимой от времени цикла ПЛК, с использованием единого системного времени.
// ==============================================================================



IF IN THEN
    IF NOT L_Running THEN
        L_Start_Time := VI_System_Time_MS;
        L_Running := TRUE;
        ET := T#0s;
        Q := FALSE;
    ELSE
        // Обработка переполнения UDINT (примерно 49 дней)
        ET := TO_TIME((SEL(VI_System_Time_MS >= L_Start_Time, VI_System_Time_MS - L_Start_Time, (4294967295 - L_Start_Time) + VI_System_Time_MS + 1)));
        
        IF ET >= PT THEN
            Q := TRUE;
            ET := PT;
        ELSE
            Q := FALSE;
        END_IF;
    END_IF;
ELSE
    L_Running := FALSE;
    ET := T#0s;
    Q := FALSE;
END_IF;
// >>> BULK_SYNC_ANCHOR: FB_System_Timer <<<
          
END_FUNCTION_BLOCK

FUNCTION_BLOCK FB_NVRAM_Manager
  VAR_INPUT
    VI_Command : BYTE;
    VI_Offset : UDINT;
    VI_DataRef : REFERENCE TO BYTE;
    VI_DataSize : UDINT;
    VI_System_Time_MS : UDINT;
    VI_Operator_ID : STRING(10);
    VI_IsActivePLC : BOOL;
    VI_TwoPersonConfirmation : BOOL;
  END_VAR
  VAR_OUTPUT
    VO_Done : BOOL;
    VO_Error : BOOL;
    VO_ErrorID : UDINT;
    VO_HMI_Status_Message : STRING(200);
  END_VAR
  VAR
    L_prev_Command : BYTE;
    L_cmd_rising : BOOL;
    L_i : UDINT;
    L_Data_Changed : BOOL;
    L_pData : POINTER TO BYTE;
  END_VAR
  VAR CONSTANT
    C_MAX_NVRAM_SIZE : UDINT := 12800;
  END_VAR

            // Детекция фронта команды
L_cmd_rising := (VI_Command <> 0) AND (L_prev_Command = 0);
L_prev_Command := VI_Command;

IF L_cmd_rising THEN
    VO_Done := FALSE;
    VO_Error := FALSE;
    VO_ErrorID := 0;
    VO_HMI_Status_Message := '';
    
    // Валидация смещения
    IF VI_Offset >= C_MAX_NVRAM_SIZE THEN
        VO_Error := TRUE;
        VO_ErrorID := 16#1501;
        VO_HMI_Status_Message := 'NVRAM: Неверное смещение';
        VO_Done := TRUE;
        RETURN;
    END_IF;

    // Валидация указателя
    IF NOT __ISVALIDREF(VI_DataRef) THEN
        VO_Error := TRUE;
        VO_ErrorID := 16#150A;
        VO_HMI_Status_Message := 'NVRAM: Недействительная ссылка на данные';
        VO_Done := TRUE;
        RETURN;
    END_IF;

    L_pData := ADR(VI_DataRef);

    IF (VI_Offset + VI_DataSize) > C_MAX_NVRAM_SIZE THEN
        VO_Error := TRUE;
        VO_ErrorID := 16#150B;
        VO_HMI_Status_Message := 'NVRAM: Размер данных превышает доступный объем';
        VO_Done := TRUE;
        RETURN;
    END_IF;

    IF VI_Command = 2 THEN
    VO_Error := TRUE;
    VO_ErrorID := 16#150D;
    VO_HMI_Status_Message := 'NVRAM: READ not implemented';
    VO_Done := TRUE;
    RETURN;
END_IF;

IF VI_Command = 1 THEN // ЗАПИСЬ (WRITE)
        IF NOT VI_IsActivePLC THEN
            VO_Error := TRUE;
            VO_ErrorID := 16#1509;
            VO_HMI_Status_Message := 'NVRAM: Запись запрещена (STANDBY)';
        ELSE
            // Проверка на изменение данных перед записью
            L_Data_Changed := FALSE;
            FOR L_i := 0 TO VI_DataSize - 1 DO
                IF GVL_Retain.G_NVRAM_Data[VI_Offset + L_i] <> L_pData[L_i] THEN
                    L_Data_Changed := TRUE;
                    EXIT;
                END_IF;
            END_FOR;
            
            IF L_Data_Changed THEN
                // Безопасное копирование (WRITE)
                FOR L_i := 0 TO VI_DataSize - 1 DO
                    GVL_Retain.G_NVRAM_Data[VI_Offset + L_i] := L_pData[L_i];
                END_FOR;
                VO_HMI_Status_Message := 'NVRAM: Данные успешно сохранены в RETAIN';
            ELSE
                VO_HMI_Status_Message := 'NVRAM: Данные не изменились, запись пропущена';
            END_IF;
        END_IF;
        VO_Done := TRUE;
    END_IF;
END_IF;

IF VI_Command = 0 THEN
    VO_Done := FALSE;
END_IF;
// >>> BULK_SYNC_ANCHOR: FB_NVRAM_Manager <<<
          
END_FUNCTION_BLOCK

FUNCTION_BLOCK FB_History_Manager
  VAR_INPUT
    VI_System_Time_MS : UDINT;
    VI_Write_Event : BOOL;
    VI_Event : ST_History_Record;
  END_VAR
  VAR_OUTPUT
    VO_Total_Events : UDINT;
  END_VAR
  VAR
    L_Prev_Write_Event : BOOL;
  END_VAR

            IF VI_Write_Event AND NOT L_Prev_Write_Event THEN
    GVL_Retain.G_History_Buffer[GVL_Retain.G_History_Write_Idx] := VI_Event;
    GVL_Retain.G_History_Buffer[GVL_Retain.G_History_Write_Idx].timestamp_ms := VI_System_Time_MS;
    
    GVL_Retain.G_History_Write_Idx := (GVL_Retain.G_History_Write_Idx MOD GVL_CONSTANTS.C_MAX_HISTORY_RECORDS) + 1;
    GVL_Retain.G_History_Total_Events := GVL_Retain.G_History_Total_Events + 1;
END_IF;
L_Prev_Write_Event := VI_Write_Event;

VO_Total_Events := GVL_Retain.G_History_Total_Events;
// >>> BULK_SYNC_ANCHOR: FB_History_Manager <<<
          
END_FUNCTION_BLOCK

FUNCTION_BLOCK FB_Heating_Manifold_Control
  VAR_INPUT
    VI_System_Time_MS : UDINT;
    VI_IsActivePLC : BOOL;
    VI_DHW_Heating_Demand : BOOL;
    VI_Freeze_Mode_Active : BOOL;
    VI_Target_Supply_Temp : REAL;
    VI_Any_Zone_Active : ARRAY[1..GVL_CONSTANTS.C_MAX_MANIFOLDS] OF BOOL;
  END_VAR
  VAR_OUTPUT
    VO_Manifold_Pumps : ARRAY[1..GVL_CONSTANTS.C_MAX_MANIFOLDS] OF BOOL;
    VO_Manifold_Valves : ARRAY[1..GVL_CONSTANTS.C_MAX_MANIFOLDS] OF REAL;
    VO_Status : ARRAY[1..GVL_CONSTANTS.C_MAX_MANIFOLDS] OF ST_Manifold_Status;
  END_VAR
  VAR_IN_OUT
    VI_Manifold_Pressures : ARRAY[1..GVL_CONSTANTS.C_MAX_MANIFOLDS] OF REAL;
    VI_Manifold_Currents : ARRAY[1..GVL_CONSTANTS.C_MAX_MANIFOLDS] OF REAL;
    VI_Manifold_Temps_Supply : ARRAY[1..GVL_CONSTANTS.C_MAX_MANIFOLDS] OF REAL;
    VI_Manifold_Temps_Return : ARRAY[1..GVL_CONSTANTS.C_MAX_MANIFOLDS] OF REAL;
  END_VAR
  VAR
    L_i : INT;
    L_Delta_T : REAL;
    L_PID_Valves : ARRAY[1..GVL_CONSTANTS.C_MAX_MANIFOLDS] OF FB_PID_Controller;
    L_PID_Timer : ARRAY[1..GVL_CONSTANTS.C_MAX_MANIFOLDS] OF FB_System_Timer;
    L_Pump_Run_Timer : ARRAY[1..GVL_CONSTANTS.C_MAX_MANIFOLDS] OF FB_System_Timer;
    L_Pump_Pause_Timer : ARRAY[1..GVL_CONSTANTS.C_MAX_MANIFOLDS] OF FB_System_Timer;
    L_Pump_In_Pause : ARRAY[1..GVL_CONSTANTS.C_MAX_MANIFOLDS] OF BOOL;
    L_Pump_Diag : ARRAY[1..GVL_CONSTANTS.C_MAX_MANIFOLDS] OF FB_Device_Predictive_Diag;
  END_VAR

            // ==============================================================================
// Heating manifold control helper
// Internal refactoring helper for FB_Heating_System_Manager.
// Valve test override remains in FB_Heating_System_Manager for now.
// ==============================================================================



FOR L_i := 1 TO GVL_CONSTANTS.C_MAX_MANIFOLDS DO
    L_PID_Timer[L_i](IN := TRUE, PT := T#1s, VI_System_Time_MS := VI_System_Time_MS);
    IF L_PID_Timer[L_i].Q THEN
        L_PID_Timer[L_i](IN := FALSE, PT := T#1s, VI_System_Time_MS := VI_System_Time_MS);
        L_PID_Timer[L_i](IN := TRUE, PT := T#1s, VI_System_Time_MS := VI_System_Time_MS);

        L_PID_Valves[L_i](
            VI_SetPoint := VI_Target_Supply_Temp,
            VI_ProcessValue := VI_Manifold_Temps_Supply[L_i],
            VI_Kp := 2.0,
            VI_Tn := 120.0,
            VI_Tv := 0.0,
            VI_Y_Min := 0.0,
            VI_Y_Max := 100.0,
            VI_Cycle_Time_S := 1.0,
            VO_Output => VO_Manifold_Valves[L_i]
        );
    END_IF;

    L_Pump_Run_Timer[L_i](
        IN := VO_Manifold_Pumps[L_i] AND NOT L_Pump_In_Pause[L_i],
        PT := T#72h,
        VI_System_Time_MS := VI_System_Time_MS
    );
    IF L_Pump_Run_Timer[L_i].Q THEN
        L_Pump_In_Pause[L_i] := TRUE;
    END_IF;

    L_Pump_Pause_Timer[L_i](
        IN := L_Pump_In_Pause[L_i],
        PT := T#1h,
        VI_System_Time_MS := VI_System_Time_MS
    );
    IF L_Pump_Pause_Timer[L_i].Q THEN
        L_Pump_In_Pause[L_i] := FALSE;
    END_IF;

    IF VI_DHW_Heating_Demand THEN
        VO_Manifold_Pumps[L_i] := FALSE;
        VO_Manifold_Valves[L_i] := 0.0;
    ELSE
        VO_Manifold_Pumps[L_i] := VI_IsActivePLC AND VI_Any_Zone_Active[L_i] AND NOT L_Pump_In_Pause[L_i];
    END_IF;

    IF VI_Freeze_Mode_Active THEN
        VO_Manifold_Pumps[L_i] := TRUE;
        IF VO_Manifold_Valves[L_i] < 35.0 THEN
            VO_Manifold_Valves[L_i] := 35.0;
        END_IF;
    END_IF;

    VO_Status[L_i].Pump_On := VO_Manifold_Pumps[L_i];
    VO_Status[L_i].Pump_Current := VI_Manifold_Currents[L_i];
    VO_Status[L_i].Pressure := VI_Manifold_Pressures[L_i];
    VO_Status[L_i].Temp_Supply := VI_Manifold_Temps_Supply[L_i];
    VO_Status[L_i].Temp_Return := VI_Manifold_Temps_Return[L_i];
    VO_Status[L_i].Valve_Pos := VO_Manifold_Valves[L_i];

    L_Pump_Diag[L_i](
        VI_Current_Value := VI_Manifold_Currents[L_i],
        VI_Nominal_Value := 0.55,
        VI_Is_Running := VO_Manifold_Pumps[L_i],
        VI_Reset_Stats := FALSE,
        VI_System_Time_MS := VI_System_Time_MS,
        VIO_Health_Data := VO_Status[L_i].Health
    );

    IF VO_Manifold_Pumps[L_i] THEN
        L_Delta_T := VI_Manifold_Temps_Supply[L_i] - VI_Manifold_Temps_Return[L_i];

        VO_Status[L_i].Error := FALSE;
        VO_Status[L_i].Error_ID := 0;

        IF VI_Manifold_Currents[L_i] <= 0.01 THEN
            VO_Status[L_i].Error := TRUE;
            VO_Status[L_i].Error_ID := TO_WORD(GVL_CONFIG.ERR_PUMP_NO_CURRENT);
        ELSIF VI_Manifold_Currents[L_i] < 0.3 THEN
            VO_Status[L_i].Error := TRUE;
            VO_Status[L_i].Error_ID := TO_WORD(GVL_CONFIG.ERR_PUMP_UNDERCURRENT);
        ELSIF VI_Manifold_Currents[L_i] > 1.5 THEN
            VO_Status[L_i].Error := TRUE;
            VO_Status[L_i].Error_ID := TO_WORD(GVL_CONFIG.ERR_PUMP_OVERCURRENT);
        END_IF;

        IF (NOT VO_Status[L_i].Error) AND ((VI_Manifold_Pressures[L_i] < 1.5) OR (VI_Manifold_Pressures[L_i] > 2.5)) THEN
            VO_Status[L_i].Error := TRUE;
            VO_Status[L_i].Error_ID := TO_WORD(GVL_CONFIG.ERR_PRESSURE_OUT_OF_RANGE);
        END_IF;

        IF NOT VO_Status[L_i].Error THEN
            IF L_Delta_T < 5.0 THEN
                VO_Status[L_i].Error := TRUE;
                VO_Status[L_i].Error_ID := TO_WORD(GVL_CONFIG.ERR_DELTA_T_LOW);
            ELSIF L_Delta_T > 10.0 THEN
                VO_Status[L_i].Error := TRUE;
                VO_Status[L_i].Error_ID := TO_WORD(GVL_CONFIG.ERR_DELTA_T_HIGH);
            END_IF;
        END_IF;
    END_IF;
END_FOR;

// >>> BULK_SYNC_ANCHOR: FB_Heating_Manifold_Control <<<
          
END_FUNCTION_BLOCK

FUNCTION_BLOCK FB_Socket_Manager
  VAR_INPUT
    VI_System_Time_MS : UDINT;
    VI_IsActivePLC : BOOL;
    VI_Scenario : E_SCENARIO_TYPE;
    VI_Fire_Alarm : BOOL;
    VI_Flood_Alarm : BOOL;
    VI_Security_Armed : BOOL;
  END_VAR
  VAR_OUTPUT
    VO_Socket_States : ARRAY[1..GVL_CONSTANTS.C_MAX_SOCKETS] OF BOOL;
    VO_Internal_States : ARRAY[1..GVL_CONSTANTS.C_MAX_SOCKETS] OF BOOL;
  END_VAR
  VAR_IN_OUT
    VI_Manual_Override : ARRAY[1..GVL_CONSTANTS.C_MAX_SOCKETS] OF BOOL;
    VI_Physical_Switches : ARRAY[1..GVL_CONSTANTS.C_MAX_SOCKETS] OF BOOL;
    VI_Rule_Actions : ARRAY[1..GVL_CONSTANTS.C_MAX_RULES] OF ST_Rule_Action;
    VI_IO_Modules_Online : ARRAY[1..GVL_CONSTANTS.C_MAX_MODULES] OF BOOL;
  END_VAR
  VAR
    L_i : INT;
    L_j : INT;
    L_Rule_State : BOOL;
    L_Rule_Active : BOOL;
    L_Internal_State : ARRAY[1..GVL_CONSTANTS.C_MAX_SOCKETS] OF BOOL;
    L_Manual_Trig : ARRAY[1..GVL_CONSTANTS.C_MAX_SOCKETS] OF R_TRIG;
  END_VAR

            // Менеджер управления розетками.
// Обеспечивает работу по сценариям, правилам и аварийное отключение (без локальных выключателей розеток).


IF NOT VI_IsActivePLC THEN RETURN; END_IF;


// Проверка связи с модулями ввода-вывода
FOR L_i := 1 TO GVL_CONSTANTS.C_MAX_MODULES DO
    IF NOT VI_IO_Modules_Online[L_i] THEN
        // Переход в безопасное состояние при потере связи (отключение всех розеток)
        FOR L_j := 1 TO GVL_CONSTANTS.C_MAX_SOCKETS DO
            VO_Socket_States[L_j] := FALSE;
        END_FOR;
        RETURN;
    END_IF;
END_FOR;

FOR L_i := 1 TO GVL_CONSTANTS.C_MAX_SOCKETS DO
    L_Rule_Active := FALSE;
    L_Rule_State := FALSE;
    
    L_Manual_Trig[L_i](CLK := VI_Manual_Override[L_i]);
    
    // Ручное переключение
    IF L_Manual_Trig[L_i].Q THEN
        L_Internal_State[L_i] := NOT L_Internal_State[L_i];
    END_IF;

    // Проверка правил для текущей розетки
    FOR L_j := 1 TO GVL_CONSTANTS.C_MAX_RULES DO
        IF VI_Rule_Actions[L_j].Active AND VI_Rule_Actions[L_j].Target_ID = L_i THEN
            IF VI_Rule_Actions[L_j].Action_Type = E_Rule_Action_Type.ACTION_SET_SOCKET THEN
                L_Rule_Active := TRUE;
                L_Rule_State := (VI_Rule_Actions[L_j].Value > 0.5);
                L_Internal_State[L_i] := L_Rule_State; // Синхронизация внутреннего состояния
            ELSIF VI_Rule_Actions[L_j].Action_Type = E_Rule_Action_Type.ACTION_TOGGLE_SOCKET AND VI_Rule_Actions[L_j].Triggered THEN
                L_Internal_State[L_i] := NOT L_Internal_State[L_i]; // Toggle
            END_IF;
        END_IF;
    END_FOR;

    // Аварийное отключение
    IF VI_Fire_Alarm OR VI_Flood_Alarm THEN
        // Розетки 1-4 неотключаемые (холодильник, сервер и т.д.)
        IF L_i > 4 THEN
            VO_Socket_States[L_i] := FALSE;
        ELSE
            // Критические розетки сохраняют свое текущее внутреннее состояние, а не форсируются в TRUE
            VO_Socket_States[L_i] := L_Internal_State[L_i];
        END_IF;
    ELSIF VI_Scenario = E_SCENARIO_TYPE.SCENARIO_AWAY OR VI_Security_Armed THEN
        // Master Off
        IF L_i > 4 THEN
            VO_Socket_States[L_i] := FALSE;
        ELSE
            // Неотключаемые розетки могут управляться вручную
            VO_Socket_States[L_i] := L_Internal_State[L_i];
        END_IF;
    ELSE
        // Нормальный режим: состояние определяется внутренним состоянием (ручным или правилом)
        IF L_Rule_Active THEN
            VO_Socket_States[L_i] := L_Rule_State;
        ELSE
            VO_Socket_States[L_i] := L_Internal_State[L_i];
        END_IF;
    END_IF;
END_FOR;

VO_Internal_States := L_Internal_State;

// >>> BULK_SYNC_ANCHOR: FB_Socket_Manager <<<
          
END_FUNCTION_BLOCK

FUNCTION_BLOCK FB_Gas_Smoke_Manager
  VAR_INPUT
    VI_System_Time_MS : UDINT;
    VI_IsActivePLC : BOOL;
    VI_Mute_Request : BOOL;
  END_VAR
  VAR_OUTPUT
    VO_Smoke_Detected : BOOL;
    VO_Gas_Detected : BOOL;
    VO_CO_Warning_Level : BOOL;
    VO_CO_Alarm_Level : BOOL;
    VO_Status_Msg : STRING(200);
  END_VAR
  VAR_IN_OUT
    VI_Methane_LEL : ARRAY[1..GVL_CONSTANTS.C_MAX_METHANE_SENSORS] OF REAL;
    VI_CO_PPM : ARRAY[1..GVL_CONSTANTS.C_MAX_CO_SENSORS] OF REAL;
    VI_Smoke_Sensors : ARRAY[1..GVL_CONSTANTS.C_MAX_SMOKE_SENSORS] OF BOOL;
  END_VAR
  VAR
    L_Methane_Max : REAL;
    L_CO_Max : REAL;
    L_Smoke_Count : UINT;
    L_Smoke_Active : BOOL;
    L_i : INT;
    L_CO_Timer_30ppm : FB_System_Timer;
    L_CO_Timer_70ppm : FB_System_Timer;
    L_CO_Timer_400ppm : FB_System_Timer;
    L_CO_Level_30 : BOOL;
    L_CO_Level_70 : BOOL;
    L_CO_Level_400 : BOOL;
    L_Smoke_Timer : ARRAY[1..GVL_CONSTANTS.C_MAX_SMOKE_SENSORS] OF FB_System_Timer;
  END_VAR

            IF NOT VI_IsActivePLC THEN RETURN; END_IF;

// Reset outputs
VO_Smoke_Detected := FALSE;
VO_Gas_Detected := FALSE;
VO_CO_Warning_Level := FALSE;
VO_CO_Alarm_Level := FALSE;
VO_Status_Msg := 'ОК';

// --- Methane ---
L_Methane_Max := 0.0;
FOR L_i := 1 TO GVL_CONSTANTS.C_MAX_METHANE_SENSORS DO
    IF VI_Methane_LEL[L_i] > L_Methane_Max THEN
        L_Methane_Max := VI_Methane_LEL[L_i];
    END_IF;
END_FOR;

IF L_Methane_Max >= 20.0 THEN
    VO_Gas_Detected := TRUE;
END_IF;

// --- CO ---
L_CO_Max := 0.0;
FOR L_i := 1 TO GVL_CONSTANTS.C_MAX_CO_SENSORS DO
    IF VI_CO_PPM[L_i] > L_CO_Max THEN
        L_CO_Max := VI_CO_PPM[L_i];
    END_IF;
END_FOR;

L_CO_Level_30 := (L_CO_Max >= 30.0);
L_CO_Level_70 := (L_CO_Max >= 70.0);
L_CO_Level_400 := (L_CO_Max >= 400.0);

L_CO_Timer_30ppm(IN := L_CO_Level_30, PT := T#8h, VI_System_Time_MS := VI_System_Time_MS);
L_CO_Timer_70ppm(IN := L_CO_Level_70, PT := T#1h, VI_System_Time_MS := VI_System_Time_MS);
L_CO_Timer_400ppm(IN := L_CO_Level_400, PT := T#15m, VI_System_Time_MS := VI_System_Time_MS);

IF L_CO_Timer_30ppm.Q THEN
    VO_CO_Warning_Level := TRUE;
END_IF;

IF L_CO_Timer_70ppm.Q OR L_CO_Timer_400ppm.Q THEN
    VO_CO_Alarm_Level := TRUE;
END_IF;

// --- Smoke ---
L_Smoke_Count := 0;
L_Smoke_Active := FALSE;

FOR L_i := 1 TO GVL_CONSTANTS.C_MAX_SMOKE_SENSORS DO
    L_Smoke_Timer[L_i](IN := VI_Smoke_Sensors[L_i], PT := T#30s, VI_System_Time_MS := VI_System_Time_MS);

    IF VI_Smoke_Sensors[L_i] THEN
        L_Smoke_Count := L_Smoke_Count + 1;
    END_IF;

    IF L_Smoke_Timer[L_i].Q OR (L_Smoke_Count >= 2) THEN
        L_Smoke_Active := TRUE;
    END_IF;
END_FOR;

IF L_Smoke_Active THEN
    VO_Smoke_Detected := TRUE;
END_IF;

// Status
IF VO_Smoke_Detected THEN
    VO_Status_Msg := 'ПОЖАР';
ELSIF VO_Gas_Detected THEN
    VO_Status_Msg := 'УТЕЧКА ГАЗА';
ELSIF VO_CO_Alarm_Level THEN
    VO_Status_Msg := 'КРИТИЧЕСКИЙ CO';
ELSIF VO_CO_Warning_Level THEN
    VO_Status_Msg := 'ПОВЫШЕННЫЙ CO';
ELSE
    VO_Status_Msg := 'ОК';
END_IF;
// >>> BULK_SYNC_ANCHOR: FB_Gas_Smoke_Manager <<<
          
END_FUNCTION_BLOCK

FUNCTION_BLOCK FB_Sensor_Analog_Processing
  VAR_INPUT
    VI_Raw_Value : WORD;
    VI_Sensor_Type : INT := 0;
    VI_Min_Scale : REAL;
    VI_Max_Scale : REAL;
    VI_Offset : REAL;
    VI_Multiplier : REAL := 1.0;
    VI_Filter_Time_MS : UDINT := GVL_CONSTANTS.C_MS_IN_SECOND;
    VI_System_Time_MS : UDINT;
    VI_Fallback_Mode : INT := 0;
    VI_Default_Value : REAL := 0.0;
  END_VAR
  VAR_OUTPUT
    VO_Value : REAL;
    VO_Error : BOOL;
    VO_Diag_Code : WORD;
  END_VAR
  VAR
    L_Scaled : REAL;
    L_Filtered : REAL;
    L_History : ARRAY[0..9] OF REAL;
    L_History_Idx : INT := 0;
    L_History_Sum : REAL := 0.0;
    L_History_Count : INT := 0;
    L_Last_Time : UDINT;
    L_DT : UDINT;
    L_First_Scan : BOOL := TRUE;
    L_i : INT;
  END_VAR

            // 1. Error checking and scaling based on sensor type
VO_Error := FALSE;
VO_Diag_Code := 0;

CASE VI_Sensor_Type OF
    0: // 4-20mA (NAMUR NE43: < 3.6mA or > 21mA)
        IF VI_Raw_Value < GVL_CONSTANTS.C_ANALOG_3_6MA_RAW THEN // < 3.6mA (Open circuit)
            VO_Error := TRUE;
            VO_Diag_Code := 1;
        ELSIF VI_Raw_Value > GVL_CONSTANTS.C_ANALOG_21MA_RAW THEN // > 21mA (Short circuit)
            VO_Error := TRUE;
            VO_Diag_Code := 2;
        ELSE
            // 4mA = 5529, 20mA = 27648
            L_Scaled := VI_Min_Scale + (TO_REAL(VI_Raw_Value - GVL_CONSTANTS.C_ANALOG_4MA_RAW) / TO_REAL(GVL_CONSTANTS.C_ANALOG_RAW_MAX - GVL_CONSTANTS.C_ANALOG_4MA_RAW)) * (VI_Max_Scale - VI_Min_Scale);
        END_IF;
        
    1: // 0-10V (0-27648)
        IF VI_Raw_Value > GVL_CONSTANTS.C_ANALOG_10V_MAX_RAW THEN // Out of range
            VO_Error := TRUE;
            VO_Diag_Code := 3;
        ELSE
            L_Scaled := VI_Min_Scale + (TO_REAL(VI_Raw_Value) / TO_REAL(GVL_CONSTANTS.C_ANALOG_RAW_MAX)) * (VI_Max_Scale - VI_Min_Scale);
        END_IF;
        
    2: // PT100/1000 (Direct temperature * 10, e.g., 255 = 25.5C)
        // Typically, 16-bit signed integer for temperature
        IF VI_Raw_Value = 16#7FFF OR VI_Raw_Value = 16#8000 THEN // Sensor error codes
            VO_Error := TRUE;
            VO_Diag_Code := 1;
        ELSE
            L_Scaled := TO_REAL(TO_INT(VI_Raw_Value)) / 10.0;
            IF L_Scaled < VI_Min_Scale OR L_Scaled > VI_Max_Scale THEN
                VO_Error := TRUE;
                VO_Diag_Code := 3;
            END_IF;
        END_IF;
        
    ELSE
        VO_Error := TRUE;
        VO_Diag_Code := 16#FFFF; // Unknown sensor type
END_CASE;

// 2. Fallback handling
IF VO_Error THEN
    IF VI_Fallback_Mode = 1 THEN
        VO_Value := VI_Default_Value;
    END_IF;
    // If VI_Fallback_Mode = 0, VO_Value retains its last good value (L_Filtered)
    RETURN;
END_IF;

// 3. Calibration
L_Scaled := (L_Scaled * VI_Multiplier) + VI_Offset;

// 4. Moving Average Filter (ТЗ 1.2)
IF L_First_Scan THEN
    L_Filtered := L_Scaled;
    L_First_Scan := FALSE;
    L_Last_Time := VI_System_Time_MS;
    
    // Инициализация массива истории
    FOR L_i := 0 TO 9 DO
        L_History[L_i] := L_Scaled;
    END_FOR;
    L_History_Sum := L_Scaled * 10.0;
    L_History_Count := 10;
    L_History_Idx := 0;
END_IF;

L_DT := (SEL(VI_System_Time_MS >= L_Last_Time, VI_System_Time_MS - L_Last_Time, (4294967295 - L_Last_Time) + VI_System_Time_MS + 1));
IF VI_Filter_Time_MS = 0 THEN
    L_Filtered := L_Scaled;
    L_Last_Time := VI_System_Time_MS;
ELSIF L_DT >= (VI_Filter_Time_MS / 10) THEN // Обновляем 10 раз за время фильтрации
    // Вычитаем старое значение
    L_History_Sum := L_History_Sum - L_History[L_History_Idx];
    
    // Добавляем новое значение
    L_History[L_History_Idx] := L_Scaled;
    L_History_Sum := L_History_Sum + L_Scaled;
    
    // Сдвигаем индекс
    L_History_Idx := (L_History_Idx + 1) MOD 10;
    
    // Вычисляем среднее
    L_Filtered := L_History_Sum / 10.0;
    
    L_Last_Time := VI_System_Time_MS;
END_IF;

VO_Value := L_Filtered;
          
END_FUNCTION_BLOCK

FUNCTION_BLOCK FB_PLC_Heartbeat
  VAR_INPUT
    VI_Local_ID : BYTE;
    VI_System_Time : UDINT;
    VI_Remote_Pulse : BOOL;
    VI_Remote_Is_Active : BOOL;
    VI_Gateway_Ping_OK : BOOL;
  END_VAR
  VAR_OUTPUT
    VO_Is_Active : BOOL;
    VO_RTT_MS : UDINT;
    VO_Loss_Count : UDINT;
    VO_Max_RTT : UDINT;
  END_VAR
  VAR
    L_Last_Pulse : BOOL;
    L_Last_Pulse_Time : UDINT;
    L_Timeout : UDINT := 500;
    L_Pulse_Send_Time : UDINT;
    L_Last_Loss_Time : UDINT;
    L_Elapsed_Time : UDINT;
  END_VAR

            // Вспомогательная функция для безопасного вычисления разницы времени
L_Elapsed_Time := (VI_System_Time - L_Last_Pulse_Time);

// 1. Мониторинг "сердцебиения" и расчет сетевых задержек (ТЗ 8.4)
IF VI_Remote_Pulse <> L_Last_Pulse THEN
    // Вычисляем время между изменениями сигнала
    VO_RTT_MS := L_Elapsed_Time;
    // Фиксируем пиковые задержки для диагностики сети
    IF VO_RTT_MS > VO_Max_RTT THEN VO_Max_RTT := VO_RTT_MS; END_IF;
    L_Last_Pulse := VI_Remote_Pulse;
    L_Last_Pulse_Time := VI_System_Time;
    L_Elapsed_Time := 0; // Сбрасываем после обновления
END_IF;

// Подсчет статистики потерь связи (ТЗ 8.4)
IF L_Elapsed_Time > L_Timeout THEN
    IF (VI_System_Time - L_Last_Loss_Time) >= 1000 THEN
        VO_Loss_Count := VO_Loss_Count + 1;
        L_Last_Loss_Time := VI_System_Time;
    END_IF;
ELSE
    L_Last_Loss_Time := VI_System_Time;
END_IF;

// 2. Логика определения роли (Active/Standby) и предотвращение Split-Brain (ТЗ 8.3)
// Уровень 1: Проверка наличия связи с партнером
IF L_Elapsed_Time < L_Timeout THEN
    // Связь есть: Договариваемся о ролях на основе приоритета ID
    IF VI_Local_ID = 1 THEN
        VO_Is_Active := TRUE; // ПЛК А всегда активен при наличии связи
    ELSE
        VO_Is_Active := NOT VI_Remote_Is_Active; // ПЛК B активен только если А не активен
    END_IF;
ELSE
    // Связи нет: Пытаемся определить, кто из нас "живее"
    // Уровень 3: Если связи с партнером нет, проверяем доступность внешнего шлюза
    IF VI_Local_ID = 1 THEN
        // ПЛК А становится активным всегда при потере связи с партнером (fallback)
        VO_Is_Active := TRUE;
    ELSE
        // ПЛК B ждет таймаут удержания роли (2 секунды), прежде чем стать активным
        IF L_Elapsed_Time >= 2000 THEN
            // ПЛК B берет управление если он видит шлюз, а связи с А нет.
            // Если шлюз недоступен, B ждет дольше (fallback).
            IF VI_Gateway_Ping_OK THEN
                VO_Is_Active := TRUE;
            ELSIF L_Elapsed_Time >= 5000 THEN
                VO_Is_Active := TRUE; // Fallback: ПЛК А мертв и шлюз мертв
            ELSE
                VO_Is_Active := FALSE;
            END_IF;
        ELSE
            VO_Is_Active := FALSE;
        END_IF;
    END_IF;
END_IF;
          
END_FUNCTION_BLOCK

FUNCTION_BLOCK FB_Smoke_Detector
  VAR_INPUT
    VI_Smoke_Signal : BOOL;
  END_VAR
  VAR_OUTPUT
    VO_Smoke_Detected : BOOL;
  END_VAR

            VO_Smoke_Detected := VI_Smoke_Signal;
          
END_FUNCTION_BLOCK

FUNCTION_BLOCK FB_Simulation_Manager
  VAR_INPUT
    VI_System_Time_MS : UDINT;
    VI_IsActivePLC : BOOL;
    VI_Scenario : E_SCENARIO_TYPE;
    VI_Config : ST_Scenario_Config;
  END_VAR
  VAR_OUTPUT
    VO_Sim_Lights : ARRAY[1..32] OF BOOL;
    VO_Sim_Active : BOOL;
    VO_Sim_Water_Leak : ARRAY[1..GVL_CONSTANTS.C_MAX_FLOOD_SENSORS] OF BOOL;
    VO_Sim_Gas_Leak : ARRAY[1..GVL_CONSTANTS.C_MAX_METHANE_SENSORS] OF REAL;
  END_VAR
  VAR
    L_Random : FB_Random_Generator;
    L_Last_Toggle : UDINT;
    L_i : INT;
    L_Rand_Val : UDINT;
    L_Test_Mode : BOOL := FALSE;
  END_VAR

            IF VI_Scenario = E_SCENARIO_TYPE.SCENARIO_AWAY AND VI_Config.Presence_Simulation_Enabled THEN
    VO_Sim_Active := TRUE;
    
    // Переключаем свет каждые 30 минут
    IF (VI_System_Time_MS - L_Last_Toggle) >= (GVL_CONSTANTS.C_MS_IN_MINUTE * 30) THEN
        L_Last_Toggle := VI_System_Time_MS;
        
        FOR L_i := 1 TO 32 DO
            L_Rand_Val := 1;
            VO_Sim_Lights[L_i] := (L_Rand_Val > 80); // 20% шанс включения
        END_FOR;
    END_IF;
ELSE
    VO_Sim_Active := FALSE;
    FOR L_i := 1 TO 32 DO VO_Sim_Lights[L_i] := FALSE; END_FOR;
END_IF;

// Симуляция аварий в тестовом режиме
IF L_Test_Mode THEN
    // Генерация случайных протечек (очень редко)
    L_Rand_Val := 1;
    IF L_Rand_Val = 42 THEN
        VO_Sim_Water_Leak[1] := TRUE;
    END_IF;
    
    // Симуляция утечки газа
    L_Rand_Val := 1;
    IF L_Rand_Val = 77 THEN
        VO_Sim_Gas_Leak[1] := 15.0; // 15% LEL
    END_IF;
ELSE
    FOR L_i := 1 TO GVL_CONSTANTS.C_MAX_FLOOD_SENSORS DO VO_Sim_Water_Leak[L_i] := FALSE; END_FOR;
    FOR L_i := 1 TO GVL_CONSTANTS.C_MAX_METHANE_SENSORS DO VO_Sim_Gas_Leak[L_i] := 0.0; END_FOR;
END_IF;
// >>> BULK_SYNC_ANCHOR: FB_Simulation_Manager <<<
          
END_FUNCTION_BLOCK

FUNCTION_BLOCK FB_System_Health_Orchestrator
  VAR_OUTPUT
    VO_First_Fault_Active : BOOL;
    VO_First_Fault_Type : INT;
    VO_First_Fault_Source : INT;
    VO_System_Severity : E_System_Severity;
    VO_Root_Cause : E_System_Root_Cause;
    VO_Watchdog_Fault : BOOL;
  END_VAR
  VAR
    fbSafety : FB_Safety_Manager;
    fbWatchdog : FB_Watchdog;
    fbSystemHealth : FB_System_Health;
    fbStateManager : FB_State_Manager;
    fbHMIInterface : FB_HMI_Interface;
    fbFaultLogger : FB_Fault_Logger;
  END_VAR

            // ==============================================================================
// System health orchestrator helper
//
// Internal helper for PRG_System.
// Owns safety latch update, watchdog, system health aggregation,
// system mode calculation, HMI/fault publication, diagnostic exports,
// and human-readable mode/cause text projection.
// ==============================================================================



fbSafety(
    VI_Gas_Alarm := GVL_STATE.G_Safety_Gas_Alarm,
    VI_Leak_Alarm := GVL_STATE.G_Safety_Leak_Alarm,
    VI_Smoke_Alarm := GVL_STATE.G_Safety_Smoke_Alarm,
    VI_Reset := GVL_COMMAND.G_Reset_Errors,
    VO_Gas_Latched => GVL_STATE.G_Safety_Gas_Latched,
    VO_Leak_Latched => GVL_STATE.G_Safety_Leak_Latched,
    VO_Smoke_Latched => GVL_STATE.G_Safety_Smoke_Latched,
    VO_Emergency_Stop => GVL_STATE.G_Safety_Emergency_Stop
);

GVL_STATE.G_Freeze_Hardware_Degraded := GVL_STATUS.G_Diagnostics.Backup_Pump_Fault OR GVL_STATUS.G_Diagnostics.Electric_Heater_Fault;
GVL_STATE.G_Freeze_Hardware_Failed := GVL_STATUS.G_Diagnostics.Backup_Pump_Fault AND GVL_STATUS.G_Diagnostics.Electric_Heater_Fault;

fbWatchdog(
    VI_System_Time_MS := GVL_STATUS.G_System_Time_MS
);

fbSystemHealth(
    VI_Smoke_Detected := GVL_HEALTH_BRIDGE.G_Smoke_Detected OR GVL_STATE.G_Safety_Smoke_Latched,
    VI_Gas_Detected := GVL_HEALTH_BRIDGE.G_Gas_Detected OR GVL_STATE.G_Safety_Gas_Latched,
    VI_CO_Warning_Level := GVL_HEALTH_BRIDGE.G_CO_Warning_Level,
    VI_CO_Alarm_Level := GVL_HEALTH_BRIDGE.G_CO_Alarm_Level,
    VI_Leak_Detected := GVL_HEALTH_BRIDGE.G_Leak_Detected OR GVL_STATE.G_Safety_Leak_Latched,
    VI_Sensor_Fault := GVL_STATE.G_Heating_Sensor_Fault OR GVL_STATE.G_DHW_Sensor_Fault OR GVL_STATUS.G_Diagnostics.Manifold_Pressure_Fault_Active OR GVL_STATUS.G_Diagnostics.Manifold_Current_Fault_Active OR GVL_STATUS.G_Diagnostics.Manifold_Return_Temp_Fault_Active,
    VI_IO_Offline := GVL_STATE.G_Heating_IO_Fault OR GVL_STATE.G_DHW_IO_Fault OR GVL_STATE.G_Ventilation_IO_Fault OR GVL_STATE.G_Lighting_IO_Fault,
    VI_Comm_Fault := GVL_STATE.G_Access_Comm_Fault,
    VI_Watchdog_Fault := fbWatchdog.VO_Watchdog_Fault,
    VI_Subsystem_Fault := GVL_STATE.G_Heating_Subsystem_Degraded OR GVL_STATE.G_DHW_Subsystem_Degraded OR GVL_STATE.G_Ventilation_Subsystem_Degraded OR GVL_STATUS.G_Diagnostics.Manifold_Pressure_Fault_Active OR GVL_STATUS.G_Diagnostics.Manifold_Current_Fault_Active OR GVL_STATUS.G_Diagnostics.Manifold_Return_Temp_Fault_Active
);

fbStateManager(
    VI_System_Severity := fbSystemHealth.VO_System_Severity,
    VI_Root_Cause := fbSystemHealth.VO_Root_Cause,
    VI_Freeze_Risk := GVL_STATE.G_Safety_Freeze_Risk
);

fbHMIInterface(
    VI_Severity := fbSystemHealth.VO_System_Severity,
    VI_RootCause := fbSystemHealth.VO_Root_Cause,
    VI_Status_Msg := fbStateManager.VO_Status_Msg
);

fbFaultLogger(
    VI_Severity := fbSystemHealth.VO_System_Severity,
    VI_RootCause := fbSystemHealth.VO_Root_Cause,
    VI_Time_MS := GVL_STATUS.G_System_Time_MS
);

GVL_STATUS.G_System_Mode_Msg := fbStateManager.VO_Status_Msg;

GVL_STATUS.G_Diagnostics.Sensor_Fault :=
    GVL_STATE.G_Heating_Sensor_Fault OR
    GVL_STATE.G_DHW_Sensor_Fault OR
    GVL_STATUS.G_Diagnostics.Manifold_Pressure_Fault_Active OR
    GVL_STATUS.G_Diagnostics.Manifold_Current_Fault_Active OR
    GVL_STATUS.G_Diagnostics.Manifold_Return_Temp_Fault_Active;

GVL_STATUS.G_Diagnostics.IO_Offline :=
    GVL_STATE.G_Heating_IO_Fault OR
    GVL_STATE.G_DHW_IO_Fault OR
    GVL_STATE.G_Ventilation_IO_Fault OR
    GVL_STATE.G_Lighting_IO_Fault;

GVL_STATUS.G_Diagnostics.Subsystem_Degraded :=
    GVL_STATE.G_Heating_Subsystem_Degraded OR
    GVL_STATE.G_DHW_Subsystem_Degraded OR
    GVL_STATE.G_Ventilation_Subsystem_Degraded OR
    GVL_STATUS.G_Diagnostics.Manifold_Pressure_Fault_Active OR
    GVL_STATUS.G_Diagnostics.Manifold_Current_Fault_Active OR
    GVL_STATUS.G_Diagnostics.Manifold_Return_Temp_Fault_Active;

GVL_GATEWAY.G_Gateway_HMI_Status_Message := fbHMIInterface.VO_HMI_Status_Text;
IF fbFaultLogger.VO_Last_Event_Text <> '' THEN
    GVL_HEALTH_BRIDGE.G_Last_Fault_Event_Text := fbFaultLogger.VO_Last_Event_Text;
END_IF;

GVL_STATE.G_System_Mode := fbStateManager.VO_System_Mode;

CASE GVL_STATE.G_System_Mode OF
    E_System_Operating_Mode.MODE_SAFE_STOP:
        GVL_STATE.G_System_Mode_Text := 'SAFE_STOP';

    E_System_Operating_Mode.MODE_FREEZE_PROTECTION:
        GVL_STATE.G_System_Mode_Text := 'FREEZE_PROTECTION';

    E_System_Operating_Mode.MODE_DEGRADED:
        GVL_STATE.G_System_Mode_Text := 'DEGRADED';

    ELSE
        GVL_STATE.G_System_Mode_Text := 'NORMAL';
END_CASE;

CASE fbSystemHealth.VO_Root_Cause OF
    E_System_Root_Cause.ROOT_FIRE:
        GVL_STATUS.G_System_Mode_Cause := 'Пожар/дым';
    E_System_Root_Cause.ROOT_GAS_LEAK:
        GVL_STATUS.G_System_Mode_Cause := 'Утечка газа';
    E_System_Root_Cause.ROOT_CO_CRITICAL:
        GVL_STATUS.G_System_Mode_Cause := 'Критический CO';
    E_System_Root_Cause.ROOT_CO_WARNING:
        GVL_STATUS.G_System_Mode_Cause := 'Повышенный CO';
    E_System_Root_Cause.ROOT_WATER_LEAK:
        GVL_STATUS.G_System_Mode_Cause := 'Протечка воды';
    E_System_Root_Cause.ROOT_WATCHDOG_FAULT:
        GVL_STATUS.G_System_Mode_Cause := 'Ошибка watchdog';
    E_System_Root_Cause.ROOT_IO_OFFLINE:
        GVL_STATUS.G_System_Mode_Cause := 'Недоступен модуль IO';
    E_System_Root_Cause.ROOT_COMM_FAULT:
        GVL_STATUS.G_System_Mode_Cause := 'Ошибка связи';
    E_System_Root_Cause.ROOT_SENSOR_FAULT:
        GVL_STATUS.G_System_Mode_Cause := 'Ошибка датчика';
    E_System_Root_Cause.ROOT_SUBSYSTEM_FAULT:
        GVL_STATUS.G_System_Mode_Cause := 'Ошибка подсистемы';
    ELSE
        GVL_STATUS.G_System_Mode_Cause := 'Аварийные режимы отсутствуют';
END_CASE;

VO_First_Fault_Active := fbSystemHealth.VO_First_Fault_Active;
VO_First_Fault_Type := fbSystemHealth.VO_First_Fault_Type;
VO_First_Fault_Source := fbSystemHealth.VO_First_Fault_Source;
VO_System_Severity := fbSystemHealth.VO_System_Severity;
VO_Root_Cause := fbSystemHealth.VO_Root_Cause;
VO_Watchdog_Fault := fbWatchdog.VO_Watchdog_Fault;

GVL_STATUS.G_System_Mode_Msg := fbStateManager.VO_Status_Msg;

// >>> BULK_SYNC_ANCHOR: FB_System_Health_Orchestrator <<<
          
END_FUNCTION_BLOCK

FUNCTION_BLOCK FB_Boiler_OpenTherm_Interface
  VAR_INPUT
    VI_Enable : ARRAY[1..GVL_CONSTANTS.C_MAX_BOILERS] OF BOOL;
    VI_Setpoint : ARRAY[1..GVL_CONSTANTS.C_MAX_BOILERS] OF REAL;
    VI_OT_Online : ARRAY[1..GVL_CONSTANTS.C_MAX_BOILERS] OF BOOL;
    VI_OT_Error : ARRAY[1..GVL_CONSTANTS.C_MAX_BOILERS] OF BOOL;
  END_VAR
  VAR_OUTPUT
    VO_OT_Enable : ARRAY[1..GVL_CONSTANTS.C_MAX_BOILERS] OF BOOL;
    VO_OT_Setpoint : ARRAY[1..GVL_CONSTANTS.C_MAX_BOILERS] OF REAL;
    VO_OT_Command_Valid : ARRAY[1..GVL_CONSTANTS.C_MAX_BOILERS] OF BOOL;
  END_VAR
  VAR
    L_i : INT;
  END_VAR

            FOR L_i := 1 TO GVL_CONSTANTS.C_MAX_BOILERS DO
    VO_OT_Enable[L_i] := FALSE;
    VO_OT_Setpoint[L_i] := 0.0;
    VO_OT_Command_Valid[L_i] := FALSE;

    IF VI_Enable[L_i] AND VI_OT_Online[L_i] AND NOT VI_OT_Error[L_i] THEN
        VO_OT_Enable[L_i] := TRUE;
        VO_OT_Setpoint[L_i] := LIMIT(20.0, VI_Setpoint[L_i], 80.0);
        VO_OT_Command_Valid[L_i] := TRUE;
    END_IF;
END_FOR;
          
END_FUNCTION_BLOCK

FUNCTION_BLOCK FB_PID_Controller
  VAR_INPUT
    VI_SetPoint : REAL;
    VI_ProcessValue : REAL;
    VI_Kp : REAL;
    VI_Tn : REAL;
    VI_Tv : REAL;
    VI_Y_Min : REAL := 0.0;
    VI_Y_Max : REAL := 100.0;
    VI_Manual_Mode : BOOL;
    VI_Manual_Value : REAL;
    VI_Deadband : REAL := 0.1;
    VI_Cycle_Time_S : REAL := 0.01;
    VI_Reset : BOOL;
  END_VAR
  VAR_OUTPUT
    VO_Output : REAL;
    VO_Error : REAL;
    VO_Limiting : BOOL;
  END_VAR
  VAR
    L_Integral_Sum : REAL;
    L_Prev_Error : REAL;
    L_Derivative : REAL;
    L_Output_Raw : REAL;
  END_VAR

            // Расчет ошибки
VO_Error := VI_SetPoint - VI_ProcessValue;

// Проверка мертвой зоны
IF ABS(VO_Error) < VI_Deadband THEN
    VO_Error := 0.0;
END_IF;

IF VI_Reset THEN
    L_Integral_Sum := 0.0;
    L_Prev_Error := 0.0;
    VO_Output := 0.0;
    RETURN;
END_IF;

IF VI_Manual_Mode THEN
    VO_Output := VI_Manual_Value;
    // Безударный переход: при выходе из ручного режима выход должен остаться прежним.
    // Так как Выход = P + I + D, то I = Выход - P - D.
    // Для простоты D при переходе обнуляем (или игнорируем), тогда I = Выход - P.
    L_Integral_Sum := VO_Output - (VI_Kp * VO_Error);
    L_Prev_Error := VO_Error;
    RETURN;
END_IF;

// Пропорциональная составляющая
L_Output_Raw := VI_Kp * VO_Error;

// Интегральная составляющая (Метод трапеций)
IF VI_Tn > 0.0 THEN
    // Anti-windup: не накапливаем интеграл, если выход уже на пределе и ошибка того же знака
    IF NOT VO_Limiting OR (VO_Error > 0.0 AND L_Output_Raw < VI_Y_Max) OR (VO_Error < 0.0 AND L_Output_Raw > VI_Y_Min) THEN
        L_Integral_Sum := L_Integral_Sum + (VI_Kp / VI_Tn) * VO_Error * VI_Cycle_Time_S;
    END_IF;
    L_Output_Raw := L_Output_Raw + L_Integral_Sum;
END_IF;

// Дифференциальная составляющая
IF VI_Tv > 0.0 THEN
    L_Derivative := (VO_Error - L_Prev_Error) / VI_Cycle_Time_S;
    L_Output_Raw := L_Output_Raw + VI_Kp * VI_Tv * L_Derivative;
END_IF;

L_Prev_Error := VO_Error;

// Ограничение выхода
IF L_Output_Raw > VI_Y_Max THEN
    VO_Output := VI_Y_Max;
    VO_Limiting := TRUE;
ELSIF L_Output_Raw < VI_Y_Min THEN
    VO_Output := VI_Y_Min;
    VO_Limiting := TRUE;
ELSE
    VO_Output := L_Output_Raw;
    VO_Limiting := FALSE;
END_IF;
// >>> BULK_SYNC_ANCHOR: FB_PID_Controller <<<
          
END_FUNCTION_BLOCK

FUNCTION_BLOCK FB_Boiler_Cascade_Manager
  VAR_INPUT
    VI_Enable : BOOL;
    VI_System_Time_MS : UDINT;
    VI_Boiler_Stop : BOOL;
    VI_DHW_Heating_Demand : BOOL;
    VI_DHW_Target_Temp : REAL;
    VI_Target_Supply_Temp : REAL;
    VI_Demand_Power : REAL;
    VI_Boiler_Flame_Status : ARRAY[1..GVL_CONSTANTS.C_MAX_BOILERS] OF BOOL;
    VI_Boiler_Error_Status : ARRAY[1..GVL_CONSTANTS.C_MAX_BOILERS] OF BOOL;
    VI_Boiler_OT_Online : ARRAY[1..GVL_CONSTANTS.C_MAX_BOILERS] OF BOOL;
    VI_Boiler_Modulation : ARRAY[1..GVL_CONSTANTS.C_MAX_BOILERS] OF REAL;
  END_VAR
  VAR_OUTPUT
    VO_Boiler_Enable : ARRAY[1..GVL_CONSTANTS.C_MAX_BOILERS] OF BOOL;
    VO_Boiler_Setpoint : ARRAY[1..GVL_CONSTANTS.C_MAX_BOILERS] OF REAL;
    VO_Lead_Boiler : BYTE;
  END_VAR
  VAR
    L_i : INT;
    L_Lead_Boiler : BYTE := 1;
    L_Last_Rotation_MS : UDINT := 0;
    L_Rotation_Initialized : BOOL := FALSE;
    L_Rotation_Period_MS : UDINT := 604800000;
    L_Lead_Available : BOOL;
    L_Reserve_Available : BOOL;
    L_Reserve_Boiler : BYTE;
    L_Start_Reserve : BOOL;
    L_Target_Setpoint : REAL;
    L_Flame_Miss_Timer : ARRAY[1..GVL_CONSTANTS.C_MAX_BOILERS] OF TON;
  END_VAR

            // Сброс выходов по умолчанию
FOR L_i := 1 TO GVL_CONSTANTS.C_MAX_BOILERS DO
    VO_Boiler_Enable[L_i] := FALSE;
    VO_Boiler_Setpoint[L_i] := 0.0;
END_FOR;

// Инициализация ротации
IF NOT L_Rotation_Initialized THEN
    L_Last_Rotation_MS := VI_System_Time_MS;
    L_Rotation_Initialized := TRUE;
END_IF;

// Принудительная остановка
IF VI_Boiler_Stop THEN
    VO_Lead_Boiler := L_Lead_Boiler;
    RETURN;
END_IF;

// Ротация строго каждые 168 часов
IF (VI_System_Time_MS - L_Last_Rotation_MS) >= L_Rotation_Period_MS THEN
    IF GVL_CONSTANTS.C_MAX_BOILERS > 1 THEN
        L_Lead_Boiler := 3 - L_Lead_Boiler;
    END_IF;
    L_Last_Rotation_MS := VI_System_Time_MS;
END_IF;

L_Reserve_Boiler := SEL(L_Lead_Boiler = 1, 1, 2);

L_Lead_Available :=
    VI_Boiler_OT_Online[L_Lead_Boiler] AND
    NOT VI_Boiler_Error_Status[L_Lead_Boiler];

L_Reserve_Available :=
    (GVL_CONSTANTS.C_MAX_BOILERS > 1) AND
    VI_Boiler_OT_Online[L_Reserve_Boiler] AND
    NOT VI_Boiler_Error_Status[L_Reserve_Boiler];

// Контроль "команда есть, пламени нет" для ведущего котла
L_Flame_Miss_Timer[L_Lead_Boiler](
    IN := VI_Enable AND L_Lead_Available AND NOT VI_DHW_Heating_Demand AND NOT VI_Boiler_Flame_Status[L_Lead_Boiler],
    PT := T#120s
);

IF L_Flame_Miss_Timer[L_Lead_Boiler].Q AND L_Reserve_Available THEN
    L_Lead_Boiler := L_Reserve_Boiler;
    L_Last_Rotation_MS := VI_System_Time_MS;
    L_Lead_Available :=
        VI_Boiler_OT_Online[L_Lead_Boiler] AND
        NOT VI_Boiler_Error_Status[L_Lead_Boiler];
    L_Reserve_Boiler := SEL(L_Lead_Boiler = 1, 1, 2);
    L_Reserve_Available :=
        (GVL_CONSTANTS.C_MAX_BOILERS > 1) AND
        VI_Boiler_OT_Online[L_Reserve_Boiler] AND
        NOT VI_Boiler_Error_Status[L_Reserve_Boiler];
END_IF;

// Нет запроса тепла
IF NOT VI_Enable THEN
    VO_Lead_Boiler := L_Lead_Boiler;
    RETURN;
END_IF;

// Целевая уставка
IF VI_DHW_Heating_Demand THEN
    L_Target_Setpoint := LIMIT(20.0, VI_DHW_Target_Temp + 15.0, 85.0);
ELSE
    L_Target_Setpoint := LIMIT(20.0, VI_Target_Supply_Temp + 5.0, 80.0);
END_IF;

// Выбор ведущего по доступности
IF NOT L_Lead_Available AND L_Reserve_Available THEN
    L_Lead_Boiler := L_Reserve_Boiler;
    L_Lead_Available := TRUE;
    L_Reserve_Boiler := SEL(L_Lead_Boiler = 1, 1, 2);
    L_Reserve_Available :=
        (GVL_CONSTANTS.C_MAX_BOILERS > 1) AND
        VI_Boiler_OT_Online[L_Reserve_Boiler] AND
        NOT VI_Boiler_Error_Status[L_Reserve_Boiler];
END_IF;

// Основной котёл
IF L_Lead_Available THEN
    VO_Boiler_Enable[L_Lead_Boiler] := TRUE;
    VO_Boiler_Setpoint[L_Lead_Boiler] := L_Target_Setpoint;
END_IF;

// Резервный котёл: >80% или отказ основного
L_Start_Reserve :=
    L_Reserve_Available AND
    (
        (VI_Demand_Power > 80.0) OR
        (NOT L_Lead_Available)
    );

IF L_Start_Reserve THEN
    VO_Boiler_Enable[L_Reserve_Boiler] := TRUE;
    VO_Boiler_Setpoint[L_Reserve_Boiler] := L_Target_Setpoint;
END_IF;

VO_Lead_Boiler := L_Lead_Boiler;
          
END_FUNCTION_BLOCK

FUNCTION_BLOCK FB_Ownership_Watchdog
  VAR_INPUT
    VI_Gas_Level : REAL;
    VI_Gas_Alarm : BOOL;
    VI_Leak_Alarm : BOOL;
    VI_Smoke_Alarm : BOOL;
  END_VAR
  VAR_OUTPUT
    VO_Ownership_Violation : BOOL;
  END_VAR
  VAR
    L_Last_Gas_Alarm : BOOL;
    L_Last_Leak_Alarm : BOOL;
    L_Last_Smoke_Alarm : BOOL;
  END_VAR

            VO_Ownership_Violation := FALSE;

// Gas: signal present, alarm disappeared
IF (VI_Gas_Level > 20.0) AND L_Last_Gas_Alarm AND (NOT VI_Gas_Alarm) THEN
    VO_Ownership_Violation := TRUE;
END_IF;

// Leak: once latched should not drop instantly
IF L_Last_Leak_Alarm AND (NOT VI_Leak_Alarm) THEN
    VO_Ownership_Violation := TRUE;
END_IF;

// Smoke: same rule
IF L_Last_Smoke_Alarm AND (NOT VI_Smoke_Alarm) THEN
    VO_Ownership_Violation := TRUE;
END_IF;

L_Last_Gas_Alarm := VI_Gas_Alarm;
L_Last_Leak_Alarm := VI_Leak_Alarm;
L_Last_Smoke_Alarm := VI_Smoke_Alarm;
          
END_FUNCTION_BLOCK

FUNCTION_BLOCK FB_System_Scenario_Arbitration
  VAR_INPUT
    VI_System_Time_MS : UDINT;
    VI_IsActivePLC : BOOL;
    VI_System_Mode : E_System_Operating_Mode;
    VI_Security_Armed : BOOL;
  END_VAR
  VAR_IN_OUT
    VIO_Scenario_Req_Operator : E_SCENARIO_TYPE;
    VIO_Scenario_Req_Gateway : E_SCENARIO_TYPE;
    VIO_Scenario_Req_Rule : E_SCENARIO_TYPE;
    VIO_Scenario_Req_Final : E_SCENARIO_TYPE;
    VIO_Scenario_Intent : E_SCENARIO_TYPE;
    VIO_Scenario_Source : E_SCENARIO_SOURCE;
  END_VAR
  VAR
    fbLogEvent : FB_LogEvent;
    fbScenarioManager : FB_Scenario_Manager;
  END_VAR

            // ==============================================================================
// System scenario arbitration helper
//
// Internal helper for PRG_System.
// Owns scenario request validation, priority resolution, fail-safe clamp,
// degraded-mode adaptation, policy logging, and FB_Scenario_Manager call.
// ==============================================================================



// === SCENARIO REQUEST VALIDATION ===
// Normalize invalid values to NONE to avoid corrupt inputs.
// Actual enum range in E_SCENARIO_TYPE is 0..7.
IF TO_USINT(VIO_Scenario_Req_Operator) > 7 THEN
    VIO_Scenario_Req_Operator := E_SCENARIO_TYPE.SCENARIO_NONE;
END_IF;

IF TO_USINT(VIO_Scenario_Req_Gateway) > 7 THEN
    VIO_Scenario_Req_Gateway := E_SCENARIO_TYPE.SCENARIO_NONE;
END_IF;

IF TO_USINT(VIO_Scenario_Req_Rule) > 7 THEN
    VIO_Scenario_Req_Rule := E_SCENARIO_TYPE.SCENARIO_NONE;
END_IF;

// === SCENARIO PRIORITY RESOLUTION ===
// Produces VIO_Scenario_Req_Final (TRACE ONLY, not executed directly)
IF VI_System_Mode = E_System_Operating_Mode.MODE_SAFE_STOP THEN
    VIO_Scenario_Req_Final := 0;
    VIO_Scenario_Source := SRC_SAFETY;
ELSIF VIO_Scenario_Req_Operator <> 0 THEN
    VIO_Scenario_Req_Final := VIO_Scenario_Req_Operator;
    VIO_Scenario_Source := SRC_OPERATOR;
ELSIF VIO_Scenario_Req_Gateway <> 0 THEN
    VIO_Scenario_Req_Final := VIO_Scenario_Req_Gateway;
    VIO_Scenario_Source := SRC_GATEWAY;
ELSIF VIO_Scenario_Req_Rule <> 0 THEN
    VIO_Scenario_Req_Final := VIO_Scenario_Req_Rule;
    VIO_Scenario_Source := SRC_RULE;
ELSE
    VIO_Scenario_Req_Final := GVL_STATUS.G_Current_Scenario;
    VIO_Scenario_Source := SRC_NONE;
END_IF;

VIO_Scenario_Intent := VIO_Scenario_Req_Final;

// === FAIL-SAFE SCENARIO CLAMP ===
CASE VI_System_Mode OF
    E_System_Operating_Mode.MODE_SAFE_STOP:
        VIO_Scenario_Intent := E_SCENARIO_TYPE.SCENARIO_NONE;

    E_System_Operating_Mode.MODE_FREEZE_PROTECTION:
        VIO_Scenario_Intent := E_SCENARIO_TYPE.SCENARIO_NONE;

    E_System_Operating_Mode.MODE_DEGRADED:
        CASE VIO_Scenario_Intent OF
            E_SCENARIO_TYPE.SCENARIO_NONE,
            E_SCENARIO_TYPE.SCENARIO_PRESENCE,
            E_SCENARIO_TYPE.SCENARIO_AWAY,
            E_SCENARIO_TYPE.SCENARIO_SLEEP:
                ; // allowed in degraded
        ELSE
            VIO_Scenario_Intent := E_SCENARIO_TYPE.SCENARIO_NONE;
        END_CASE;
END_CASE;

// === CONTEXT FAIL-SAFE AUTOMATION ===
// If security is armed and no explicit source is requesting another scenario,
// force safe occupancy context to AWAY while system remains in MODE_NORMAL.
IF VI_System_Mode = E_System_Operating_Mode.MODE_NORMAL THEN
    IF VI_Security_Armed AND
       (VIO_Scenario_Req_Operator = E_SCENARIO_TYPE.SCENARIO_NONE) AND
       (VIO_Scenario_Req_Gateway = E_SCENARIO_TYPE.SCENARIO_NONE) AND
       (VIO_Scenario_Req_Rule = E_SCENARIO_TYPE.SCENARIO_NONE) AND
       (VIO_Scenario_Intent <> E_SCENARIO_TYPE.SCENARIO_AWAY) THEN

        IF VIO_Scenario_Intent <> E_SCENARIO_TYPE.SCENARIO_AWAY THEN
            VIO_Scenario_Intent := E_SCENARIO_TYPE.SCENARIO_AWAY;
            VIO_Scenario_Source := SRC_POLICY;

            fbLogEvent(
                VI_Event_Type := 5,
                VI_Timestamp := VI_System_Time_MS,
                VI_Param1 := TO_UDINT(VIO_Scenario_Source),
                VI_Param2 := TO_UDINT(E_SCENARIO_TYPE.SCENARIO_AWAY)
            );
        END_IF;
    END_IF;
END_IF;

// === DEGRADED-AWARE SCENARIO ADAPTATION ===
// Soft adaptation in degraded mode: keep explicit requests intact,
// but if no source is requesting a scenario, move behavior to a safer baseline.
IF VI_System_Mode = E_System_Operating_Mode.MODE_DEGRADED THEN
    IF (VIO_Scenario_Req_Operator = E_SCENARIO_TYPE.SCENARIO_NONE) AND
       (VIO_Scenario_Req_Gateway = E_SCENARIO_TYPE.SCENARIO_NONE) AND
       (VIO_Scenario_Req_Rule = E_SCENARIO_TYPE.SCENARIO_NONE) THEN

        IF VI_Security_Armed THEN
            IF VIO_Scenario_Intent <> E_SCENARIO_TYPE.SCENARIO_AWAY THEN
                VIO_Scenario_Intent := E_SCENARIO_TYPE.SCENARIO_AWAY;
                VIO_Scenario_Source := SRC_POLICY;

                fbLogEvent(
                    VI_Event_Type := 6,
                    VI_Timestamp := VI_System_Time_MS,
                    VI_Param1 := TO_UDINT(VIO_Scenario_Source),
                    VI_Param2 := TO_UDINT(E_SCENARIO_TYPE.SCENARIO_AWAY)
                );
            END_IF;

        ELSIF VIO_Scenario_Intent = E_SCENARIO_TYPE.SCENARIO_PRESENCE THEN
            IF VIO_Scenario_Intent <> E_SCENARIO_TYPE.SCENARIO_SLEEP THEN
                VIO_Scenario_Intent := E_SCENARIO_TYPE.SCENARIO_SLEEP;
                VIO_Scenario_Source := SRC_POLICY;

                fbLogEvent(
                    VI_Event_Type := 7,
                    VI_Timestamp := VI_System_Time_MS,
                    VI_Param1 := TO_UDINT(VIO_Scenario_Source),
                    VI_Param2 := TO_UDINT(E_SCENARIO_TYPE.SCENARIO_SLEEP)
                );
            END_IF;
        END_IF;
    END_IF;
END_IF;

fbScenarioManager(
    VI_System_Time_MS := VI_System_Time_MS,
    VI_Activate_Request := VIO_Scenario_Intent,
    VI_IsActivePLC := VI_IsActivePLC,
    VI_System_Mode := VI_System_Mode,
    VO_Current_Scenario => GVL_STATUS.G_Current_Scenario
);

// >>> BULK_SYNC_ANCHOR: FB_System_Scenario_Arbitration <<<
          
END_FUNCTION_BLOCK

FUNCTION_BLOCK FB_Redundancy_Manager
  VAR_INPUT
    VI_System_Time_MS : UDINT;
    VI_Local_PLC_ID : BYTE;
    VI_Remote_Pulse : BOOL;
    VI_Remote_Is_Active : BOOL;
    VI_Gateway_Ping_OK : BOOL;
    VI_Remote_State : ST_System_State_Snapshot;
    VI_Local_State : ST_System_State_Snapshot;
  END_VAR
  VAR_OUTPUT
    VO_Local_Role : E_PLC_ROLE;
    VO_Local_Pulse : BOOL;
    VO_Sync_Data_Req : BOOL;
    VO_Status_Msg : STRING(200);
    VO_Synced_State : ST_System_State_Snapshot;
    VO_State_Updated : BOOL;
  END_VAR
  VAR
    L_Heartbeat : FB_PLC_Heartbeat;
    L_Pulse_Timer : FB_System_Timer;
    L_Pulse_State : BOOL;
    L_Prev_Role : E_PLC_ROLE;
    L_State_Replicator : FB_State_Replication;
  END_VAR

            // 1. Генерация собственного пульса (меандр 100 мс)
L_Pulse_Timer(IN := NOT L_Pulse_Timer.Q, PT := T#100ms, VI_System_Time_MS := VI_System_Time_MS);
IF L_Pulse_Timer.Q THEN
    L_Pulse_State := NOT L_Pulse_State;
END_IF;
VO_Local_Pulse := L_Pulse_State;

// 2. Определение роли через Heartbeat
L_Heartbeat(
    VI_Local_ID := VI_Local_PLC_ID,
    VI_System_Time := VI_System_Time_MS,
    VI_Remote_Pulse := VI_Remote_Pulse,
    VI_Remote_Is_Active := VI_Remote_Is_Active,
    VI_Gateway_Ping_OK := VI_Gateway_Ping_OK
);

IF L_Heartbeat.VO_Is_Active THEN
    VO_Local_Role := E_PLC_ROLE.ROLE_ACTIVE;
    VO_Status_Msg := 'ПЛК АКТИВЕН (ВЕДУЩИЙ)';
ELSE
    VO_Local_Role := E_PLC_ROLE.ROLE_STANDBY;
    VO_Status_Msg := 'ПЛК В РЕЗЕРВЕ (ВЕДОМЫЙ)';
END_IF;

// 3. Запрос на синхронизацию при переходе в ACTIVE
IF VO_Local_Role = E_PLC_ROLE.ROLE_ACTIVE AND L_Prev_Role = E_PLC_ROLE.ROLE_STANDBY THEN
    VO_Sync_Data_Req := TRUE;
ELSE
    VO_Sync_Data_Req := FALSE;
END_IF;

L_State_Replicator(
    VI_Local_Role := VO_Local_Role,
    VI_Sync_Req := VO_Sync_Data_Req,
    VI_Local_State := VI_Local_State,
    VI_Remote_State := VI_Remote_State,
    VI_System_Time_MS := VI_System_Time_MS
);
VO_Synced_State := L_State_Replicator.VO_Synced_State;
VO_State_Updated := L_State_Replicator.VO_State_Updated;

L_Prev_Role := VO_Local_Role;
// >>> BULK_SYNC_ANCHOR: FB_Redundancy_Manager <<<
          
END_FUNCTION_BLOCK

FUNCTION_BLOCK FB_IO_Module_Watchdog
  VAR_INPUT
    VI_System_Time_MS : UDINT;
    VI_Module_ID : BYTE;
    VI_Heartbeat_Signal : BOOL;
    VI_Timeout_MS : UDINT := 2000;
  END_VAR
  VAR_OUTPUT
    VO_Module_Online : BOOL;
    VO_Error_Active : BOOL;
  END_VAR
  VAR
    L_Last_Heartbeat_State : BOOL;
    L_Last_Heartbeat_Time : UDINT;
    L_Elapsed_Time : UDINT;
  END_VAR

            // Отслеживание изменения сигнала
IF VI_Heartbeat_Signal <> L_Last_Heartbeat_State THEN
    L_Last_Heartbeat_Time := VI_System_Time_MS;
    L_Last_Heartbeat_State := VI_Heartbeat_Signal;
END_IF;

// Проверка таймаута
L_Elapsed_Time := (SEL(VI_System_Time_MS >= L_Last_Heartbeat_Time, VI_System_Time_MS - L_Last_Heartbeat_Time, (4294967295 - L_Last_Heartbeat_Time) + VI_System_Time_MS + 1));

IF L_Elapsed_Time > VI_Timeout_MS THEN
    VO_Module_Online := FALSE;
    VO_Error_Active := TRUE;
ELSE
    VO_Module_Online := TRUE;
    VO_Error_Active := FALSE;
END_IF;
// >>> BULK_SYNC_ANCHOR: FB_IO_Module_Watchdog <<<
          
END_FUNCTION_BLOCK

FUNCTION_BLOCK FB_System_Evacuation
  VAR
    L_i : INT;
  END_VAR

            // ==============================================================================
// System evacuation helper
//
// Internal helper for PRG_System.
// Owns evacuation guidance, target/hazard zone name projection,
// and evacuation lighting activation.
// ==============================================================================



FOR L_i := 1 TO 32 DO
    GVL_STATE.G_Evac_Guidance[L_i] := 0;

    IF GVL_STATE.G_Evac_Hazard_Zone[L_i] THEN
        GVL_STATE.G_Evac_Guidance[L_i] := -1;
    END_IF;

    IF GVL_CONFIG.G_Evac_Exit_Zones[L_i] AND NOT GVL_STATE.G_Evac_Hazard_Zone[L_i] THEN
        GVL_STATE.G_Evac_Guidance[L_i] := 1;
    END_IF;
END_FOR;

GVL_STATUS.G_Evac_Target_Zone_Name := '';
GVL_STATUS.G_Evac_Hazard_Zone_Name := '';

FOR L_i := 1 TO 32 DO
    IF (GVL_STATUS.G_Evac_Hazard_Zone_Name = '') AND GVL_STATE.G_Evac_Hazard_Zone[L_i] THEN
        GVL_STATUS.G_Evac_Hazard_Zone_Name := GVL_CONFIG.G_Evac_Zone_Names[L_i];
        IF GVL_STATUS.G_Evac_Hazard_Zone_Name = '' THEN
            GVL_STATUS.G_Evac_Hazard_Zone_Name := CONCAT('Zone ', INT_TO_STRING(L_i));
        END_IF;
    END_IF;

    IF (GVL_STATUS.G_Evac_Target_Zone_Name = '') AND (GVL_STATE.G_Evac_Guidance[L_i] = 1) THEN
        GVL_STATUS.G_Evac_Target_Zone_Name := GVL_CONFIG.G_Evac_Zone_Names[L_i];
        IF GVL_STATUS.G_Evac_Target_Zone_Name = '' THEN
            GVL_STATUS.G_Evac_Target_Zone_Name := CONCAT('Zone ', INT_TO_STRING(L_i));
        END_IF;
    END_IF;
END_FOR;

IF GVL_STATE.G_System_Mode = E_System_Operating_Mode.MODE_SAFE_STOP AND GVL_STATE.G_Safety_Smoke_Latched THEN
    GVL_STATE.G_Evacuation_Lighting_Active := TRUE;
ELSE
    GVL_STATE.G_Evacuation_Lighting_Active := FALSE;
END_IF;

// >>> BULK_SYNC_ANCHOR: FB_System_Evacuation <<<
          
END_FUNCTION_BLOCK

FUNCTION_BLOCK FB_TwoFactor_Auth
  VAR_INPUT
    VI_System_Time_MS : UDINT;
    VI_Start_Auth : BOOL;
    VI_Method : E_TwoFactor_Method;
    VI_User_Code : STRING(6);
    VI_Reset_Success : BOOL;
  END_VAR
  VAR_OUTPUT
    VO_State : ST_TwoFactor_Auth_State;
    VO_Send_Code_Req : BOOL;
    VO_Code_To_Send : STRING(6);
  END_VAR
  VAR
    L_Generated_Code : STRING(6) := '';
    L_Start_Time : UDINT;
    R_Trig_Start : R_TRIG;
    L_Prev_User_Code : STRING(6);
    L_Lockout_Start_Time : UDINT;
    fbHMAC : FB_HMAC_SHA1;
    L_Elapsed_Time : UDINT;
    L_Time_Step : UDINT;
    L_Message : ARRAY[0..7] OF BYTE;
    L_Key : ARRAY[0..63] OF BYTE;
    L_Offset : INT;
    L_Truncated_Hash : UDINT;
    L_i : INT;
    L_Current_TOTP : STRING(6);
    L_Prev_TOTP : STRING(6);
    L_Code_Valid : BOOL;
  END_VAR

            R_Trig_Start(CLK := VI_Start_Auth);

IF VI_Reset_Success THEN
    VO_State.Is_Success := FALSE;
END_IF;

IF R_Trig_Start.Q AND NOT VO_State.is_pending AND NOT VO_State.Is_Locked THEN
    VO_State.is_pending := TRUE;
    VO_State.Auth_Method := VI_Method;
    L_Start_Time := VI_System_Time_MS;
    VO_State.Attempts_Left := 3;
    VO_State.Is_Success := FALSE;
    VO_State.Is_Locked := FALSE;
    L_Prev_User_Code := '';
    
    IF VI_Method <> E_TwoFactor_Method.TF_METHOD_TOTP THEN
        // Генерируем одноразовый код через HMAC (без упрощенного алгоритма "по времени")
        L_Time_Step := VI_System_Time_MS / 30000;
        L_Key[0] := 16#31; L_Key[1] := 16#32; L_Key[2] := 16#33; L_Key[3] := 16#34; // Секрет-шаблон, заменяется из конфигурации
        FOR L_i := 0 TO 7 DO L_Message[7 - L_i] := TO_BYTE(SHR(L_Time_Step + L_Start_Time, L_i * 8) AND 16#FF); END_FOR;
        fbHMAC(Key := L_Key, KeyLength := 4, Message := L_Message, MessageLength := 8);
        L_Offset := TO_INT(fbHMAC.Hash[19] AND 16#0F);
        L_Truncated_Hash := (SHL(TO_UDINT(fbHMAC.Hash[L_Offset] AND 16#7F), 24) OR SHL(TO_UDINT(fbHMAC.Hash[L_Offset+1] AND 16#FF), 16) OR SHL(TO_UDINT(fbHMAC.Hash[L_Offset+2] AND 16#FF), 8) OR TO_UDINT(fbHMAC.Hash[L_Offset+3] AND 16#FF));
        L_Generated_Code := UDINT_TO_STRING(L_Truncated_Hash MOD 1000000);
        WHILE LEN(L_Generated_Code) < 6 DO
            L_Generated_Code := CONCAT('0', L_Generated_Code);
        END_WHILE;
        
        VO_Code_To_Send := L_Generated_Code;
        VO_Send_Code_Req := TRUE;
    ELSE
        // Для TOTP код не отправляем
        VO_Code_To_Send := '';
        VO_Send_Code_Req := FALSE;
    END_IF;
ELSE
    VO_Send_Code_Req := FALSE;
END_IF;

IF VO_State.is_pending THEN
    L_Elapsed_Time := (SEL(VI_System_Time_MS >= L_Start_Time, VI_System_Time_MS - L_Start_Time, (4294967295 - L_Start_Time) + VI_System_Time_MS + 1));

    IF L_Elapsed_Time < (GVL_CONSTANTS.C_MS_IN_MINUTE * 5) THEN
        VO_State.Time_Left_S := TO_UINT(((GVL_CONSTANTS.C_MS_IN_MINUTE * 5) - L_Elapsed_Time) / 1000);
    ELSE
        VO_State.Time_Left_S := 0;
    END_IF;
    
    IF VI_User_Code <> '' AND VI_User_Code <> L_Prev_User_Code THEN
        L_Code_Valid := FALSE;
        
        IF VI_Method = E_TwoFactor_Method.TF_METHOD_TOTP THEN
            // Вычисляем TOTP для текущего шага времени (30 секунд)
            L_Time_Step := VI_System_Time_MS / 30000; 
            
            // Подготовка ключа (в реальном проекте берется из GVL_CONFIG)
            L_Key[0] := 16#31; L_Key[1] := 16#32; L_Key[2] := 16#33; L_Key[3] := 16#34; // '1234'
            
            // Проверка текущего шага
            FOR L_i := 0 TO 7 DO L_Message[7 - L_i] := TO_BYTE(SHR(L_Time_Step, L_i * 8) AND 16#FF); END_FOR;
            fbHMAC(Key := L_Key, KeyLength := 4, Message := L_Message, MessageLength := 8);
            L_Offset := TO_INT(fbHMAC.Hash[19] AND 16#0F);
            L_Truncated_Hash := (SHL(TO_UDINT(fbHMAC.Hash[L_Offset] AND 16#7F), 24) OR SHL(TO_UDINT(fbHMAC.Hash[L_Offset+1] AND 16#FF), 16) OR SHL(TO_UDINT(fbHMAC.Hash[L_Offset+2] AND 16#FF), 8) OR TO_UDINT(fbHMAC.Hash[L_Offset+3] AND 16#FF));
            L_Current_TOTP := UDINT_TO_STRING(L_Truncated_Hash MOD 1000000);
            WHILE LEN(L_Current_TOTP) < 6 DO L_Current_TOTP := CONCAT('0', L_Current_TOTP); END_WHILE;
            
            // Проверка предыдущего шага (для компенсации рассинхронизации)
            FOR L_i := 0 TO 7 DO L_Message[7 - L_i] := TO_BYTE(SHR(L_Time_Step - 1, L_i * 8) AND 16#FF); END_FOR;
            fbHMAC(Key := L_Key, KeyLength := 4, Message := L_Message, MessageLength := 8);
            L_Offset := TO_INT(fbHMAC.Hash[19] AND 16#0F);
            L_Truncated_Hash := (SHL(TO_UDINT(fbHMAC.Hash[L_Offset] AND 16#7F), 24) OR SHL(TO_UDINT(fbHMAC.Hash[L_Offset+1] AND 16#FF), 16) OR SHL(TO_UDINT(fbHMAC.Hash[L_Offset+2] AND 16#FF), 8) OR TO_UDINT(fbHMAC.Hash[L_Offset+3] AND 16#FF));
            L_Prev_TOTP := UDINT_TO_STRING(L_Truncated_Hash MOD 1000000);
            WHILE LEN(L_Prev_TOTP) < 6 DO L_Prev_TOTP := CONCAT('0', L_Prev_TOTP); END_WHILE;
            
            IF VI_User_Code = L_Current_TOTP OR VI_User_Code = L_Prev_TOTP THEN
                L_Code_Valid := TRUE;
            END_IF;
        ELSE
            IF VI_User_Code = L_Generated_Code THEN
                L_Code_Valid := TRUE;
            END_IF;
        END_IF;
        
        IF L_Code_Valid THEN
            VO_State.Is_Success := TRUE;
            VO_State.is_pending := FALSE;
        ELSE
            IF VO_State.Attempts_Left > 0 THEN
                VO_State.Attempts_Left := VO_State.Attempts_Left - 1;
            END_IF;
            
            IF VO_State.Attempts_Left = 0 THEN
                VO_State.Is_Locked := TRUE;
                VO_State.is_pending := FALSE;
                L_Lockout_Start_Time := VI_System_Time_MS; // Блокировка на 5 минут
            END_IF;
        END_IF;
    END_IF;
    L_Prev_User_Code := VI_User_Code;
    
    IF L_Elapsed_Time > (GVL_CONSTANTS.C_MS_IN_MINUTE * 5) THEN
        VO_State.is_pending := FALSE; // Таймаут
    END_IF;
END_IF;

IF VO_State.Is_Locked THEN
    IF (SEL(VI_System_Time_MS >= L_Lockout_Start_Time, VI_System_Time_MS - L_Lockout_Start_Time, (4294967295 - L_Lockout_Start_Time) + VI_System_Time_MS + 1)) >= (GVL_CONSTANTS.C_MS_IN_MINUTE * 5) THEN
        VO_State.Is_Locked := FALSE;
    END_IF;
END_IF;
          
END_FUNCTION_BLOCK

FUNCTION_BLOCK FB_Calibration_Manager
  VAR_INPUT
    VI_Raw_Value : REAL;
    VI_Type : BYTE;
    VI_Calib_Record : ST_Sensor_Calibration_Record;
    VI_System_Time_MS : UDINT;
    VI_Start_Verification : BOOL;
  END_VAR
  VAR_OUTPUT
    VO_Calibrated_Value : REAL;
    VO_Verification_Active : BOOL;
    VO_Verification_Failed : BOOL;
    VO_Deviation_Percent : REAL;
  END_VAR
  VAR
    L_Verification_Timer : FB_System_Timer;
    L_Initial_Value : REAL;
  END_VAR

            // 1. Расчет калиброванного значения
CASE VI_Type OF
    1: VO_Calibrated_Value := VI_Raw_Value + VI_Calib_Record.offset;
    2, 3: VO_Calibrated_Value := (VI_Raw_Value * VI_Calib_Record.multiplier) + VI_Calib_Record.offset;
END_CASE;

// 2. Верификация через 1 час (ТЗ 9.5)
IF VI_Start_Verification AND NOT VO_Verification_Active THEN
    VO_Verification_Active := TRUE;
    L_Initial_Value := VO_Calibrated_Value;
END_IF;

L_Verification_Timer(IN := VO_Verification_Active, PT := T#1h, VI_System_Time_MS := VI_System_Time_MS);

IF L_Verification_Timer.Q THEN
    VO_Verification_Active := FALSE;
    
    // ТЗ 9.5: Отклонение ≤2.0% (норма) / >5.0% (ошибка)
    IF L_Initial_Value <> 0 THEN
        VO_Deviation_Percent := ABS(VO_Calibrated_Value - L_Initial_Value) / L_Initial_Value * 100.0;
    ELSE
        VO_Deviation_Percent := 0.0;
    END_IF;
    
    VO_Verification_Failed := (VO_Deviation_Percent > 5.0);
END_IF;
          
END_FUNCTION_BLOCK

FUNCTION_BLOCK FB_System_Gateway_Intent
  VAR_INPUT
    VI_System_Time_MS : UDINT;
    VI_IsActivePLC : BOOL;
    VI_Gateway_Writes_Allowed : BOOL;
  END_VAR
  VAR_IN_OUT
    VIO_FloorHeating_Temps : ARRAY[1..8] OF REAL;
    VIO_Zone_Valve_States : ARRAY[1..8] OF BOOL;
    VIO_Lighting_Base_Levels : ARRAY[1..32] OF BYTE;
    VIO_Scenario_Req_Gateway : E_SCENARIO_TYPE;
  END_VAR
  VAR
    fbGateway : FB_Gateway_Interface;
  END_VAR

            // ==============================================================================
// System gateway intent helper
//
// Internal helper for PRG_System.
// Owns gateway FB call, user intent publication, gateway command gates,
// and allowed configuration/time/scenario writes.
// ==============================================================================



fbGateway(
    VI_System_Time_MS := VI_System_Time_MS,
    VI_Local_PLC_Role := SEL(VI_IsActivePLC, E_PLC_ROLE.ROLE_STANDBY, E_PLC_ROLE.ROLE_ACTIVE),
    VI_Incoming_Command := GVL_GATEWAY.G_Gateway_Command,
    VI_Command_Received := GVL_GATEWAY.G_Gateway_Command_Received,
    VI_FloorHeating_Temps := VIO_FloorHeating_Temps,
    VI_Room_Temps := GVL_STATE.G_Room_Temps,
    VI_Zone_Valve_States := VIO_Zone_Valve_States,
    VI_Manifold_Pressures := GVL_STATE.G_Manifold_Pressures,
    VI_Manifold_Pump_States := GVL_STATE.G_Manifold_Pumps,
    VI_Outdoor_Temp := GVL_STATE.G_Outdoor_Temp,
    VI_Security_Armed := GVL_ALARM.G_Security_Armed,
    VI_Flood_Alarm_Active := GVL_ALARM.G_Flood_Alarm_Active,
    VI_Gas_Alarm_Active := GVL_ALARM.G_Gas_Alarm_Active,
    VI_Fire_Alarm_Active := GVL_ALARM.G_Fire_Alarm_Active,
    VI_Methane_Concentration := GVL_STATE.G_Methane_Sensors[1],
    VI_Lighting_Base_Levels := VIO_Lighting_Base_Levels,
    VI_Socket_States := GVL_STATE.G_Socket_States,
    VI_Blinds_Positions := GVL_STATE.G_Blinds_Positions,
    VI_Active_Scenario := GVL_STATUS.G_Current_Scenario,
    VI_Send_2FA_Req := GVL_COMMAND.G_Send_2FA_Req,
    VI_2FA_Code := GVL_COMMAND.G_2FA_Code_Out,
    VI_Allowed_IPs := GVL_CONFIG.G_Allowed_IPs,
    VO_Telegram_Msg => GVL_GATEWAY.G_Gateway_Telegram_Msg,
    VO_Send_Telegram => GVL_GATEWAY.G_Gateway_Send_Telegram,
    VO_HMI_Status_Message => GVL_GATEWAY.G_Gateway_HMI_Status_Message,

    VO_Data_Ready => GVL_GATEWAY.G_Gateway_Data_Ready,
    VO_Modbus_Registers => GVL_GATEWAY.G_Gateway_Modbus_Registers,
    VO_Arm_Req => GVL_COMMAND.G_Arm_Req,
    VO_Disarm_Req => GVL_COMMAND.G_Disarm_Req,
    VO_PIN_Code => GVL_COMMAND.G_PIN_Code,
    VO_RFID_Tag => GVL_COMMAND.G_RFID_Tag,
    VO_2FA_Code_In => GVL_COMMAND.G_2FA_Code_In,
    VO_Lighting_Override => GVL_COMMAND.G_Lighting_Override,
    VO_Blinds_Override => GVL_COMMAND.G_Blinds_Override,
    VO_Socket_Override => GVL_COMMAND.G_Socket_Override,
    VO_Reset_Errors_Req => GVL_COMMAND.G_Reset_Errors
);

GVL_INTENT_USER.I_Source_Valid := TRUE;
GVL_INTENT_USER.I_Last_Update_MS := VI_System_Time_MS;
GVL_INTENT_USER.I_Arm_Request := GVL_COMMAND.G_Arm_Req;
GVL_INTENT_USER.I_Disarm_Request := GVL_COMMAND.G_Disarm_Req;
GVL_INTENT_USER.I_PIN_Code := GVL_COMMAND.G_PIN_Code;
GVL_INTENT_USER.I_RFID_Tag := GVL_COMMAND.G_RFID_Tag;
GVL_INTENT_USER.I_2FA_Code_In := GVL_COMMAND.G_2FA_Code_In;
GVL_INTENT_USER.I_Lighting_Override_32 := GVL_COMMAND.G_Lighting_Override;
GVL_INTENT_USER.I_Blinds_Override_32 := GVL_COMMAND.G_Blinds_Override;
GVL_INTENT_USER.I_Socket_Override_32 := GVL_COMMAND.G_Socket_Override;
GVL_INTENT_USER.I_Reset_Errors := GVL_COMMAND.G_Reset_Errors;
GVL_INTENT_USER.I_Set_Temp_Req := fbGateway.VO_Set_Temp_Req;
GVL_INTENT_USER.I_Target_Zone := fbGateway.VO_Target_Zone;
GVL_INTENT_USER.I_Target_Temperature := fbGateway.VO_Target_Temp;
GVL_INTENT_USER.I_Set_Vent_Req := fbGateway.VO_Set_Vent_Req;
GVL_INTENT_USER.I_Target_Vent_Speed := fbGateway.VO_Target_Vent_Speed;
GVL_INTENT_USER.I_Set_Config_Req := fbGateway.VO_Set_Config_Req;
GVL_INTENT_USER.I_Time_Sync_Req := fbGateway.VO_Sync_Time_Req;
GVL_INTENT_USER.I_New_Time_MS := fbGateway.VO_New_Time_MS;

IF VI_Gateway_Writes_Allowed AND
   fbGateway.VO_Set_Scenario_Req AND
   ((GVL_STATE.G_System_Mode = E_System_Operating_Mode.MODE_NORMAL) OR
    (GVL_STATE.G_System_Mode = E_System_Operating_Mode.MODE_DEGRADED)) THEN
    VIO_Scenario_Req_Gateway := fbGateway.VO_Target_Scenario;
END_IF;

IF VI_Gateway_Writes_Allowed AND
   fbGateway.VO_Set_Temp_Req AND
   (GVL_STATE.G_System_Mode = E_System_Operating_Mode.MODE_NORMAL) THEN
    GVL_CONFIG.G_HMI_FloorHeating_Configs[fbGateway.VO_Target_Zone].design_temp := fbGateway.VO_Target_Temp;
END_IF;

IF VI_Gateway_Writes_Allowed AND
   fbGateway.VO_Set_Vent_Req AND
   (GVL_STATE.G_System_Mode = E_System_Operating_Mode.MODE_NORMAL) THEN
    GVL_CONFIG.G_HMI_Vent_Global_Config.default_supply_speed := fbGateway.VO_Target_Vent_Speed;
END_IF;

IF VI_Gateway_Writes_Allowed AND
   fbGateway.VO_Set_Config_Req AND
   (GVL_STATE.G_System_Mode = E_System_Operating_Mode.MODE_NORMAL) THEN
    GVL_CONFIG.G_HMI_Apply_Settings := TRUE;
END_IF;

IF VI_Gateway_Writes_Allowed AND
   fbGateway.VO_Sync_Time_Req AND
   (GVL_STATE.G_System_Mode = E_System_Operating_Mode.MODE_NORMAL) THEN
    GVL_STATUS.G_Time_Of_Day_MS := fbGateway.VO_New_Time_MS;
END_IF;

GVL_INTENT_USER.I_Scenario_Request := VIO_Scenario_Req_Gateway;
GVL_INTENT_USER.I_Gate_Open_Request := GVL_COMMAND.G_Gate_Open;
GVL_INTENT_USER.I_Wicket_Open_Request := GVL_COMMAND.G_Wicket_Open;
GVL_INTENT_USER.I_Lock_1_Open_Request := GVL_COMMAND.G_Lock_1_Open;
GVL_INTENT_USER.I_Lock_1_Close_Request := GVL_COMMAND.G_Lock_1_Close;
GVL_INTENT_USER.I_Lock_2_Open_Request := GVL_COMMAND.G_Lock_2_Open;
GVL_INTENT_USER.I_Lock_2_Close_Request := GVL_COMMAND.G_Lock_2_Close;
GVL_INTENT_USER.I_Dangerous_Action_Request := GVL_COMMAND.CMD_Dangerous_Action_Request;
GVL_INTENT_USER.I_Dangerous_Action_Confirm := GVL_COMMAND.CMD_Dangerous_Action_Confirm;
GVL_INTENT_USER.I_User_Access_Level := GVL_COMMAND.CMD_User_Access_Level;
GVL_INTENT_USER.I_Water_Selective_Recover := GVL_COMMAND.CMD_Water_Selective_Recover;
GVL_INTENT_USER.I_Gas_Selective_Recover := GVL_COMMAND.CMD_Gas_Selective_Recover;

// >>> BULK_SYNC_ANCHOR: FB_System_Gateway_Intent <<<
          
END_FUNCTION_BLOCK

FUNCTION_BLOCK FB_System_Alarm_Orchestrator
  VAR_INPUT
    VI_First_Fault_Active : BOOL;
    VI_First_Fault_Type : INT;
    VI_First_Fault_Source : INT;
  END_VAR
  VAR
    fbAlarmManager : FB_Alarm_Manager;
  END_VAR

            // ==============================================================================
// System alarm orchestrator helper
//
// Internal helper for PRG_System.
// Owns FB_Alarm_Manager call and alarm output projection.
// ==============================================================================



fbAlarmManager(
    VI_System_Time_MS := GVL_STATUS.G_System_Time_MS,
    VI_IsActivePLC := GVL_STATUS.G_Is_Active_PLC,
    VI_Gas_Alarm := GVL_ALARM.G_Gas_Alarm_Active,
    VI_Fire_Alarm := GVL_ALARM.G_Fire_Alarm_Active,
    VI_Flood_Alarm := GVL_ALARM.G_Flood_Alarm_Active,
    VI_Security_Alarm := GVL_ALARM.G_Security_Alarm,
    VI_First_Fault_Active := VI_First_Fault_Active,
    VI_First_Fault_Type := VI_First_Fault_Type,
    VI_First_Fault_Source := VI_First_Fault_Source,
    VI_Boiler_Errors := GVL_STATE.G_Boiler_Error,
    VI_Security_Msg := GVL_STATUS.G_Security_Status_Msg,
    VI_Acknowledge_All := GVL_CONFIG.G_HMI_Ack_Alarms OR GVL_COMMAND.G_Reset_Errors,
    VI_Mute_Siren := GVL_CONFIG.G_HMI_Mute_Alarm,
    VIO_Next_Alarm_ID := GVL_ALARM.G_Next_Alarm_ID,
    VO_Global_Critical => GVL_ALARM.G_Global_Critical,
    VO_Global_Warning => GVL_ALARM.G_Global_Warning,
    VO_Siren_Active => GVL_ALARM.G_Global_Siren,
    VO_Active_Count => GVL_ALARM.G_Active_Alarm_Count,
    VO_Unacked_Count => GVL_ALARM.G_Unacked_Alarm_Count,
    VO_Event_Pulse => GVL_STATUS.G_Diagnostics.Alarm_Event_Pulse,
    VO_Event_Code => GVL_STATUS.G_Diagnostics.Alarm_Event_Code,
    VO_Event_Value => GVL_STATUS.G_Diagnostics.Alarm_Event_Value,
    VO_Alarm_List => GVL_ALARM.G_Alarm_List
);

// >>> BULK_SYNC_ANCHOR: FB_System_Alarm_Orchestrator <<<
          
END_FUNCTION_BLOCK

FUNCTION_BLOCK FB_Scenario_Manager
  VAR_INPUT
    VI_Preheat_Request : BOOL;
    VI_System_Time_MS : UDINT;
    VI_Activate_Request : E_SCENARIO_TYPE;
    VI_IsActivePLC : BOOL;
    VI_System_Mode : E_System_Operating_Mode;
  END_VAR
  VAR_OUTPUT
    VO_Current_Scenario : E_SCENARIO_TYPE;
    VO_Status_Msg : STRING(200);
  END_VAR
  VAR
    L_Last_Scenario_Time : UDINT;
  END_VAR

            IF NOT VI_IsActivePLC THEN
    RETURN;
END_IF;

CASE VI_System_Mode OF
    E_System_Operating_Mode.MODE_SAFE_STOP,
    E_System_Operating_Mode.MODE_FREEZE_PROTECTION:
        IF VO_Current_Scenario <> E_SCENARIO_TYPE.SCENARIO_NONE THEN
            VO_Current_Scenario := E_SCENARIO_TYPE.SCENARIO_NONE;
            VO_Status_Msg := 'Сценарии принудительно отключены режимом безопасности';
        END_IF;
        RETURN;

    E_System_Operating_Mode.MODE_DEGRADED:
        VO_Status_Msg := 'Смена сценариев заблокирована: деградированный режим';
        RETURN;
END_CASE;

IF VI_Activate_Request <> VO_Current_Scenario THEN
    // Проверка минимального времени работы сценария
    IF (VI_System_Time_MS - L_Last_Scenario_Time) >= 60000 OR VO_Current_Scenario = E_SCENARIO_TYPE.SCENARIO_NONE THEN
        // Логика переключения сценариев
        VO_Current_Scenario := VI_Activate_Request;
        L_Last_Scenario_Time := VI_System_Time_MS;
        
        CASE VO_Current_Scenario OF
        E_SCENARIO_TYPE.SCENARIO_NONE:
            VO_Status_Msg := 'Сценарии отключены';
        E_SCENARIO_TYPE.SCENARIO_AWAY:
            VO_Status_Msg := 'Активирован сценарий: Вне дома (Охрана + Энергосбережение)';
        E_SCENARIO_TYPE.SCENARIO_SLEEP:
            VO_Status_Msg := 'Активирован сценарий: Сон (Ночное освещение + Климат)';
        E_SCENARIO_TYPE.SCENARIO_PRESENCE:
            VO_Status_Msg := 'Активирован сценарий: Имитация присутствия';
        END_CASE;
    END_IF;
END_IF;
// >>> BULK_SYNC_ANCHOR: FB_Scenario_Manager <<<


// --- PREHEAT SCENARIO INSERT ---
IF VI_Preheat_Request THEN
    // removed: direct heating write (moved to Heating Manager)
END_IF;
          
END_FUNCTION_BLOCK

FUNCTION_BLOCK FB_Heating_Adaptive_Target
  VAR_INPUT
    VI_Base_Target_Supply_Temp : REAL;
    VI_Global_Target_Temperature : REAL;
  END_VAR
  VAR_OUTPUT
    VO_Target_Supply_Temp : REAL;
    VO_Adaptive_Correction : REAL;
    VO_Adaptive_Effective_Delta : REAL;
    VO_Adaptive_Max_Delta : REAL;
  END_VAR
  VAR_IN_OUT
    VI_Zone_Configs : ARRAY[1..GVL_CONSTANTS.C_MAX_HEATING_CIRCUITS] OF ST_FloorHeating_Circuit_Config;
    VI_Floor_Temps : ARRAY[1..GVL_CONSTANTS.C_MAX_HEATING_CIRCUITS] OF REAL;
    VI_Room_Temps : ARRAY[1..16] OF REAL;
  END_VAR
  VAR
    L_Adaptive_Zone_i : INT;
    L_Adaptive_Delta : REAL;
    L_Adaptive_Weighted_Sum : REAL;
    L_Adaptive_Weight_Total : REAL;
    L_Adaptive_Weight : REAL;
  END_VAR

            // ==============================================================================
// Adaptive target calculation for heating supply temperature
//
// Internal refactoring helper for FB_Heating_System_Manager.
// The manager remains the public facade; this block only extracts the adaptive
// target calculation section to reduce large-file edit risk.
// ==============================================================================



VO_Target_Supply_Temp := VI_Base_Target_Supply_Temp;
VO_Adaptive_Max_Delta := 0.0;
L_Adaptive_Weighted_Sum := 0.0;
L_Adaptive_Weight_Total := 0.0;
VO_Adaptive_Effective_Delta := 0.0;
VO_Adaptive_Correction := 0.0;

// Global arbitration target is applied before adaptive correction.
IF VI_Global_Target_Temperature > 0.0 THEN
    VO_Target_Supply_Temp := VI_Global_Target_Temperature;
END_IF;

// Final adaptive refinement layer.
FOR L_Adaptive_Zone_i := 1 TO GVL_CONSTANTS.C_MAX_HEATING_CIRCUITS DO
    IF VI_Zone_Configs[L_Adaptive_Zone_i].zone >= 1 AND VI_Zone_Configs[L_Adaptive_Zone_i].zone <= 8 THEN
        CASE VI_Zone_Configs[L_Adaptive_Zone_i].control_type OF
            0:
                L_Adaptive_Delta :=
                    VI_Zone_Configs[L_Adaptive_Zone_i].design_temp -
                    VI_Floor_Temps[L_Adaptive_Zone_i];
                L_Adaptive_Weight := 0.6;
            1, 2:
                L_Adaptive_Delta :=
                    VI_Zone_Configs[L_Adaptive_Zone_i].design_temp -
                    VI_Room_Temps[VI_Zone_Configs[L_Adaptive_Zone_i].zone];
                L_Adaptive_Weight := 1.0;
            ELSE
                L_Adaptive_Delta :=
                    VI_Zone_Configs[L_Adaptive_Zone_i].design_temp -
                    VI_Room_Temps[VI_Zone_Configs[L_Adaptive_Zone_i].zone];
                L_Adaptive_Weight := 0.8;
        END_CASE;

